END_GET
SET
                    lSuppress := Suppress;
                  
END_SET
END_PROPERTY

PROPERTY SuppressAfterCountDown : BOOL
GET
                    SuppressAfterCountDown := lSuppressAfterCountDown;
                  
END_GET
SET
                    lSuppressAfterCountDown := SuppressAfterCountDown;
                  
END_SET
END_PROPERTY

PROPERTY SupressCountDown : UINT
GET
                    SupressCountDown := lSupressCountDown;
                  
END_GET
SET
                    lSupressCountDown := SupressCountDown;
lResolvedSuppressAfterCountDown := FALSE;

IF (SupressCountDown>0) THEN
	lSuppressAfterCountDown := TRUE;
ELSE
	lSuppressAfterCountDown := FALSE;
END_IF

                  
END_SET
END_PROPERTY

PROPERTY TypeToken : t_medium_string
GET
                    TypeToken := 'Reportable';
                  
END_GET
END_PROPERTY
END_FUNCTION_BLOCK

FUNCTION_BLOCK ReportableSet
  VAR CONSTANT
    cReportableSetMax : USINT := 16;
  END_VAR
  VAR
    lMembers : t_reportable_array;
    lCount : USINT := 0;
    lDescribeFirstContextOnly : BOOL := FALSE;
  END_VAR

            
          

METHOD clear
                  lCount := 0;
                
END_METHOD

METHOD describe
  VAR_INPUT
    executeContext : POINTER TO ExecuteContext;
  END_VAR
  VAR
    i : USINT;
  END_VAR
                  IF (executeContext^.matchOption(cExecuteOptionSyntax)) THEN
	RETURN;
END_IF

IF (executeContext^.matchOption(cExecuteOptionParameter)) THEN	
	RETURN;
END_IF

executeContext^.append(', ');
executeContext^.WriteStream^.increaseIndent();
executeContext^.formatWithNewlineIndent();
executeContext^.append('"servers": [');
executeContext^.WriteStream^.increaseIndent();

FOR i:=1 TO Count DO	
	executeContext^.recordInitiatorWithNewlineIndent();
	lMembers[i]^.describe(executeContext);
	executeContext^.recordTerminator();

	IF (lDescribeFirstContextOnly) THEN
		EXIT;
	END_IF
	
	IF (i<Count) THEN
		executeContext^.append(', ');
	END_IF
END_FOR

executeContext^.WriteStream^.decreaseIndent();
executeContext^.append(']');
executeContext^.WriteStream^.decreaseIndent();

                
END_METHOD

METHOD equals
  VAR_INPUT
    source : POINTER TO ReportableSet;
  END_VAR
  VAR
    i : USINT;
  END_VAR
                  clear();

FOR i:=1 TO source^.Count DO
	lMembers[i] := source^.Members^[i];
END_FOR

lCount := source^.Count;

                
END_METHOD

METHOD initialize
                  lCount := 0;
                
END_METHOD

METHOD insert
  VAR_INPUT
    reportable : POINTER TO t_reportable;
  END_VAR
  VAR
    i : USINT;
    ptrA : POINTER TO POINTER TO t_reportable;
    ptrB : POINTER TO POINTER TO t_reportable;
  END_VAR
                  IF (reportable=0) THEN
	RETURN;
END_IF

IF (lCount>=cReportableSetMax) THEN
	RETURN;
END_IF

IF (lCount>0) THEN
	ptrA := ADR(lMembers[1]);
	ptrB := ADR(lMembers[2]);
	FOR i:=1 TO lCount DO
		ptrA^ := ptrB^;
		ptrA := ptrA + 1;
		ptrB := ptrB + 1;
	END_FOR
END_IF

lCount := lCount + 1;
lMembers[1] := reportable;

                
END_METHOD

METHOD list
  VAR_INPUT
    stream : POINTER TO t_stream;
  END_VAR
  VAR
    i : USINT;
  END_VAR
                  stream^.increaseIndent();

FOR i:=1 TO Count DO
	stream^.indent();
	stream^.append(lMembers[i]^.lIdentity);
	stream^.newline();
END_FOR

stream^.decreaseIndent();

                
END_METHOD

METHOD pop : POINTER TO t_reportable
                  IF (lCount=0) THEN
	pop := 0;
	RETURN;
END_IF

pop := lMembers[lCount];
lCount := lCount - 1;

                
END_METHOD

METHOD push
  VAR_INPUT
    reportable : POINTER TO t_reportable;
  END_VAR
                  IF (reportable=0) THEN
	RETURN;
END_IF

IF (lCount>=cReportableSetMax) THEN
	RETURN;
END_IF

lCount := lCount + 1;
lMembers[lCount] := reportable;
                
END_METHOD

METHOD replace
  VAR_INPUT
    reportable : POINTER TO t_reportable;
  END_VAR
                  clear();
push(reportable);
                
END_METHOD

PROPERTY Count : USINT
GET
                    Count := lCount;
                  
END_GET
END_PROPERTY

PROPERTY DescribeFirstContextOnly : BOOL
GET
                    DescribeFirstContextOnly := lDescribeFirstContextOnly;
                  
END_GET
SET
                    lDescribeFirstContextOnly := DescribeFirstContextOnly;
                  
END_SET
END_PROPERTY

PROPERTY Members : POINTER TO t_reportable_array
GET
                    Members := ADR(lMembers);
                  
END_GET
END_PROPERTY
END_FUNCTION_BLOCK

FUNCTION_BLOCK ReportableState EXTENDS Reportable
  VAR
    lVRLife : ValueReferenceUDINT;
    lLife : UDINT := 2;
    lCode : t_state_code;
    lExpiringChannelMask : UINT;
    lActive : BOOL := FALSE;
    lRegistered : BOOL := FALSE;
    lSuppressPrevious : BOOL := FALSE;
    lActiveRising : BOOL := FALSE;
    lUnsuppressRising : BOOL := FALSE;
    lUnsuppressFalling : BOOL := FALSE;
    lReportedInThisInstanceCount : UDINT := 0;
    lRaisedCount : UDINT := 0;  (* lUnsuppressedInThisInstanceCount: UDINT:= 0; *)
    lRaisedTimeStep : t_timestep := 0;
    lRaisedSystemTimeMicroseconds : ULINT := 0;
    lExpiresTimeStep : t_timestep;
    lSuppressUntilExpired : BOOL := FALSE;
    lSuppressAfterExpired : BOOL := FALSE;
    lContext : t_state_context := 0;
    lContextChanged : BOOL := FALSE;
  END_VAR

            
          

METHOD clear
                  Active := FALSE;
lContext := 0;

lExpiresTimeStep := gSystemServices.Cycle.TimeStep;

                
END_METHOD

METHOD describe
  VAR_INPUT
    executeContext : POINTER TO ExecuteContext;
  END_VAR
                  SUPER^.describe(executeContext);

IF (executeContext^.matchOption(cExecuteOptionSyntax)) THEN
	executeContext^.describeSyntaxExecutable(sCommandTrigger);
	RETURN;
END_IF

IF (executeContext^.matchOption(cExecuteOptionParameter)) THEN	
	RETURN;
END_IF

executeContext^.appendPair('style','state',TRUE,TRUE);

IF (lContext<>0) THEN
	executeContext^.appendPair('context',LWORD_TO_STRING(lContext),FALSE,TRUE);
END_IF

IF (executeContext^.matchOption(cExecuteOptionVerbose)) THEN	
	executeContext^.appendPair('raised',gTypeHandler.getTokenForUDINT(RaisedCount),FALSE,TRUE);
	executeContext^.appendPair('this_instance',gTypeHandler.getTokenForUDINT(ReportedInThisInstanceCount),FALSE,TRUE);
END_IF

                
END_METHOD

METHOD initialize
                  lVRLife.initializeValueReference(lLife,NopSelf,'Life','Duration of state once triggered','timestep',cValueStyleConfigurable);

SUPER^.initialize();

lActive := FALSE;
lRegistered := FALSE;
lRaisedCount := 0;
lRaisedTimeStep := 0;
lRaisedSystemTimeMicroseconds := 0;
lExpiresTimeStep := 0;

lChannelMask := gSystemServices.ReportableChannelManager.ChannelMaskDefaultState;


                
END_METHOD

METHOD initializeState
  VAR_INPUT
    p : POINTER TO t_particle_nop;
    nme : t_token_string;
    code : t_state_code;
  END_VAR
                  lCode := code;

IF (nme='') THEN
	Name := getStringForStateCode(Code);
ELSE
	Name := nme;
END_IF

IF (p=0) THEN
	gCodeErrorHandler(pMessage:='initializing reportable with null t_particle_nop');
	RETURN;
END_IF

p^.registerNonOperational(THIS);


                
END_METHOD

METHOD raise
                  lExpiresTimeStep := gSystemServices.Cycle.TimeStep + lLife;

lActiveRising := FALSE;
lUnsuppressRising := FALSE;
lUnsuppressFalling := FALSE;

// a := a+1;

IF (NOT(Active)) THEN
	Active := TRUE;
	lActiveRising := TRUE;
	
	lReportedInThisInstanceCount := 1;
	lRaisedCount := lRaisedCount + 1;
	lRaisedTimeStep := gSystemServices.Cycle.TimeStep;
	lRaisedSystemTimeMicroseconds := gSystemServices.Cycle.SystemTimeMicroseconds;

	IF (lSuppressUntilExpired) THEN
		SupressCountDown := 1; 	
	END_IF

	(*IF (Suppress) THEN
		lUnsuppressedInThisInstanceCount := 0;
	ELSE
		lUnsuppressedInThisInstanceCount := 1;	
	END_IF*)
	
	lSuppressPrevious := lSuppress;
	
	RETURN;
END_IF

lReportedInThisInstanceCount := lReportedInThisInstanceCount + 1;

IF ((NOT(lSuppressPrevious)) AND (lSuppress)) THEN
	lUnsuppressFalling := TRUE;
END_IF

IF ((NOT(lSuppress)) AND (lSuppressPrevious)) THEN
	lUnsuppressRising := TRUE;
END_IF

lSuppressPrevious := lSuppress;

(*IF (Suppress) THEN
	lUnsuppressedInThisInstanceCount := 0;
ELSE
	lUnsuppressedInThisInstanceCount := lUnsuppressedInThisInstanceCount + 1;	
END_IF*)

                
END_METHOD

METHOD report
  VAR_INPUT
    override : BOOL;
  END_VAR
                  IF ((override) OR 
	(Override)) THEN
	RETURN;
END_IF

SUPER^.report(override);

gSystemServices.ReportableChannelManager.reportState(THIS);
                
END_METHOD

METHOD trigger
  VAR_INPUT
    override : BOOL;
  END_VAR
                  IF (override) THEN
	RETURN;
END_IF 

report(FALSE);
propagate();

                
END_METHOD

METHOD triggerWithContext
  VAR_INPUT
    context : t_state_context;
  END_VAR
                  Context := context;
trigger(FALSE);

                
END_METHOD

METHOD execute
  VAR_INPUT
    executeContext : POINTER TO ExecuteContext;
  END_VAR
                  IF (executeContext^.matchCommand(sCommandTrigger)) THEN
	trigger(FALSE);
	RETURN;
END_IF

SUPER^.execute(executeContext);

                
END_METHOD

PROPERTY Active : BOOL
GET
                    Active := lActive;

                  
END_GET
SET
                    lActive := Active;
                  
END_SET
END_PROPERTY

PROPERTY ExpiringChannelMask : UINT
GET
                    ExpiringChannelMask := lExpiringChannelMask;
                  
END_GET
SET
                    lExpiringChannelMask := ExpiringChannelMask;
                  
END_SET
END_PROPERTY

PROPERTY Code : t_state_code
GET
                    Code := lCode;

                  
END_GET
SET
                    lCode:= Code;
                  
END_SET
END_PROPERTY

PROPERTY Context : t_state_context
GET
                    Context := lContext;
                  
END_GET
SET
                    IF (lContext=Context) THEN
	RETURN;
END_IF

lContext := Context;
lContextChanged := Active;

                  
END_SET
END_PROPERTY

PROPERTY ContextChanged : BOOL
GET
                    ContextChanged:= lContextChanged;
                  
END_GET
SET
                    lContextChanged := ContextChanged;
                  
END_SET
END_PROPERTY

PROPERTY ExpiresTimeStep : t_timestep
GET
                    ExpiresTimeStep := lExpiresTimeStep;
                  
END_GET
END_PROPERTY

PROPERTY Life : UDINT
GET
                    Life := lLife;

                  
END_GET
SET
                    lLife := MAX(Life,2);

                  
END_SET
END_PROPERTY

PROPERTY RaisedCount : UDINT
GET
                    RaisedCount := lRaisedCount;
                  
END_GET
END_PROPERTY

PROPERTY RaisedTimeStep : t_timestep
GET
                    RaisedTimeStep := lRaisedTimeStep;
                  
END_GET
END_PROPERTY

PROPERTY Registered : BOOL
GET
                    Registered := lRegistered;

                  
END_GET
SET
                    IF ((lRegistered) AND (NOT(Registered)) AND (SuppressAfterExpired)) THEN
	Suppress := TRUE;
END_IF

lRegistered := Registered;
                  
END_SET
END_PROPERTY

PROPERTY ReportedInThisInstanceCount : UDINT
GET
                    ReportedInThisInstanceCount := lReportedInThisInstanceCount;
                  
END_GET
END_PROPERTY

PROPERTY SuppressAfterExpired : BOOL
GET
                    SuppressAfterExpired := lSuppressAfterExpired;
                  
END_GET
SET
                    lSuppressAfterExpired := SuppressAfterExpired;
                  
END_SET
END_PROPERTY

PROPERTY SuppressUntilExpired : BOOL
GET
                    SuppressUntilExpired := lSuppressUntilExpired;
                  
END_GET
SET
                    IF ((lSuppressUntilExpired) AND (NOT(SuppressUntilExpired))) THEN
	SuppressAfterCountDown := FALSE;
END_IF

lSuppressUntilExpired := SuppressUntilExpired;

                  
END_SET
END_PROPERTY

PROPERTY TypeToken : t_medium_string
GET
                    TypeToken := 'State';
                  
END_GET
END_PROPERTY

PROPERTY ActiveRising : BOOL
GET
                    ActiveRising := lActiveRising;
                  
END_GET
END_PROPERTY

PROPERTY Suppress : BOOL
SET
                    lSuppress := Suppress;
                  
END_SET
END_PROPERTY

PROPERTY UnsuppressFalling : BOOL
GET
                    UnsuppressFalling := lUnsuppressFalling;

                  
END_GET
END_PROPERTY

PROPERTY UnsuppressRising : BOOL
GET
                    UnsuppressRising := lUnsuppressRising;
                  
END_GET
END_PROPERTY
END_FUNCTION_BLOCK

FUNCTION_BLOCK ReportableStateManager EXTENDS Particle
  VAR CONSTANT
    cCurrentMax : UINT := 255;
  END_VAR
  VAR
    lReportableChannelManager : POINTER TO ReportableChannelManager;
    lCurrent : ARRAY[1..cCurrentMax] OF POINTER TO t_reportablestate;
    lCurrentCount : UINT := 0;
    lOverflow : BOOL := FALSE;
    a : USINT := 0;
    b : USINT := 0;
  END_VAR

            
          

METHOD clear
  VAR_INPUT
    index : UINT;
  END_VAR
  VAR
    state : POINTER TO t_reportablestate;
    i : UINT;
  END_VAR
                  IF ((index=0) OR (index>lCurrentCount)) THEN
	RETURN;
END_IF

state := lCurrent[index];

lCurrentCount := lCurrentCount - 1;
FOR i:=index TO lCurrentCount DO
	lCurrent[i] := lCurrent[i+1];
END_FOR
lCurrent[lCurrentCount+1] := 0;

IF (state=0) THEN
	RETURN;
END_IF

state^.Registered := FALSE;
lReportableChannelManager^.reportStateExpired(state);
                
END_METHOD

METHOD cycle : POINTER TO t_reportableState
  VAR_INPUT
    mask : t_channel_mask;
    cycleIndex : POINTER TO UINT;
    loop : BOOL;
  END_VAR
  VAR
    count : UINT := 0;
    state : POINTER TO t_reportableState;
  END_VAR
                  IF ((lCurrentCount=0) OR 
	(cycleIndex=0)) THEN
	cycle := 0;
	RETURN;
END_IF

IF (cycleIndex^=0) THEN
	cycle := 0;
	RETURN;
END_IF

FOR count:=1 TO lCurrentCount DO
	IF (cycleIndex^>lCurrentCount) THEN
		IF (loop) THEN
			cycleIndex^ := 1;
		ELSE
			cycleIndex^ := 0;
			cycle := 0;
			RETURN;
		END_IF
	END_IF

	state := lCurrent[cycleIndex^]; // foobar assume state is non-null
	cycleIndex^ := cycleIndex^ + 1;
	
	IF ((NOT(state^.Suppress)) AND
		(NOT(state^.Override)) AND
		(fCheckChannelMask(state^.ChannelMask,mask))) THEN
		cycle := state;
		a := a+ 1;
		RETURN;
	END_IF
END_FOR

b := b+ 1;
cycleIndex^ := 0;
cycle := 0;
                
END_METHOD

METHOD describe
  VAR_INPUT
    executeContext : POINTER TO ExecuteContext;
  END_VAR
  VAR
    i : UINT;
    str : t_stream_string;
  END_VAR
                  SUPER^.describe(executeContext);

IF (executeContext^.matchOption(cExecuteOptionSyntax)) THEN
	RETURN;
END_IF

IF (executeContext^.matchOption(cExecuteOptionParameter)) THEN	
	RETURN;
END_IF

executeContext^.append(', ');
executeContext^.WriteStream^.increaseIndent();
executeContext^.formatWithNewlineIndent();
executeContext^.append('"states": [');
executeContext^.WriteStream^.increaseIndent();

FOR i:=1 TO lCurrentCount DO	
	executeContext^.recordInitiatorWithNewlineIndent();
	lCurrent[i]^.describe(executeContext);
	executeContext^.recordTerminator();
	
	IF (i<lCurrentCount) THEN
		executeContext^.append(', ');
	END_IF
END_FOR

executeContext^.WriteStream^.decreaseIndent();
executeContext^.append(']');
executeContext^.WriteStream^.decreaseIndent();

                
END_METHOD

METHOD initialize
  VAR
    i : UINT;
  END_VAR
                  IF (lReportableChannelManager=0) THEN
	gCodeErrorHandler(pMessage:=CONCAT('null pointer in ',lIdentity));
END_IF

SUPER^.initialize();

lCurrentCount := 0;
FOR i:=1 TO cCurrentMax DO
	lCurrent[i] := 0;
END_FOR

                
END_METHOD

METHOD initializeStateManager
  VAR_INPUT
    reportableChannelManager : POINTER TO ReportableChannelManager;
  END_VAR
                  lReportableChannelManager := reportableChannelManager;

                
END_METHOD

METHOD operator
  VAR
    i : UINT;
    state : POINTER TO t_reportablestate;
  END_VAR
                  FOR i:=1 TO lCurrentCount DO
	state := lCurrent[i];
	
	IF (state^.ContextChanged) THEN
		state^.ContextChanged := FALSE;
		lReportableChannelManager^.reportStateContextChanged(state);
	END_IF
	
	IF (state^.ExpiresTimeStep<=gSystemServices.Cycle.TimeStep) THEN
		clear(i);
	END_IF
END_FOR

                
END_METHOD

METHOD raise
  VAR_INPUT
    state : POINTER TO t_reportablestate;
  END_VAR
                  IF (state=0) THEN
	RETURN;
END_IF

IF (lCurrentCount>=cCurrentMax) THEN
	state^.Registered := FALSE;
	lOverflow := TRUE;
	RETURN;	
END_IF

IF (state^.Registered) THEN
	RETURN;
END_IF

lOverflow := FALSE;

lCurrentCount := lCurrentCount + 1;
lCurrent[lCurrentCount] := state;
state^.Registered := TRUE;

                
END_METHOD

PROPERTY Overflow : BOOL
GET
                    Overflow := lOverflow;
                  
END_GET
END_PROPERTY

PROPERTY TypeToken : t_medium_string
GET
                    TypeToken := 'RepStateManager';
                  
END_GET
END_PROPERTY
END_FUNCTION_BLOCK

FUNCTION fCheckUIRValidity : BOOL
  VAR_INPUT
    uir : REFERENCE TO t_ui_reportable;
  END_VAR

            IF (NOT(uir.valid)) THEN
	fCheckUIRValidity := FALSE;
	RETURN;
END_IF

IF ((uir.subsystem>cSubSystemMax) OR
	(uir.subsystem<0)) THEN
	fCheckUIRValidity := FALSE;
	RETURN;
END_IF

IF ((uir.event>cECMax) OR
	(uir.event<0)) THEN
	fCheckUIRValidity := FALSE;
	RETURN;
END_IF

IF ((uir.state>cSCMax) OR
	(uir.state<0)) THEN
	fCheckUIRValidity := FALSE;
	RETURN;
END_IF

fCheckUIRValidity := TRUE;

          
END_FUNCTION

FUNCTION getSeverityForStateCode : t_severity
  VAR_INPUT
    code : t_state_code;
  END_VAR

            getSeverityForStateCode := cSeverityNone; //foobar missing below

CASE code OF
	cSCNone:
		getSeverityForStateCode := cSeverityNone;

	cACSteerALargeSensorDelta:
		getSeverityForStateCode := cSeverityError;

	cACSecondaryNotRunning:
		getSeverityForStateCode := cSeverityError;

	cACSecondaryNotRunningModulation:
		getSeverityForStateCode := cSeverityError;

	cACSecondaryWaiting:
		getSeverityForStateCode := cSeverityWarning;

	cACSecondaryRunStateMismatch:
		getSeverityForStateCode := cSeverityWarning;

	cACSecondaryTemperature:
		getSeverityForStateCode := cSeverityWarning;
	
	cACChannelNotGood:
		getSeverityForStateCode := cSeverityError;

	cACChannelOperationalFail:
		getSeverityForStateCode := cSeverityError;

	cACChannelNotOperational:
		getSeverityForStateCode := cSeverityError;

	cACChannelOverflow:
		getSeverityForStateCode := cSeverityWarning;

	cACChannelSlaveFailed:
		getSeverityForStateCode := cSeverityError;

	cACCANOpenSlaveNotOperational:
		getSeverityForStateCode := cSeverityError;

	cACCANOpenSlaveModulation:
		getSeverityForStateCode := cSeverityError;

	cACCANOpenSlaveAllowableUp:
		getSeverityForStateCode := cSeverityError;

	cACCANOpenMasterNotOperational:
		getSeverityForStateCode := cSeverityError;

	cACCANOpenMasterModulation:
		getSeverityForStateCode := cSeverityError;

	cACCANOpenMasterAllowableUp:
		getSeverityForStateCode := cSeverityError;
	
	cACCANOpenSlaveNoValidTransmissions:
		getSeverityForStateCode := cSeverityWarning;

	cACCANOpenSlaveNotify:
		getSeverityForStateCode := cSeverityError;

	cACCANOpenSlaveBlock:
		getSeverityForStateCode := cSeverityError;

	cACCANOpenSlaveStop:
		getSeverityForStateCode := cSeverityCritical;
		
	cACUInterfaceEstop:
		getSeverityForStateCode := cSeverityCritical;

	cACUInterfaceStop:
		getSeverityForStateCode := cSeverityCritical;

	cACUInterfaceEmgy:
		getSeverityForStateCode := cSeverityWarning;

	cACUInterfaceNotReady:
		getSeverityForStateCode := cSeverityWarning;

	cACControllerTemperatureCutback:
		getSeverityForStateCode := cSeverityWarning;

	cACMotorTemperatureCutback:
		getSeverityForStateCode := cSeverityWarning;

	cACMotorTemperatureSensor:
		getSeverityForStateCode := cSeverityError;

	cACCoolantReservoir:
		getSeverityForStateCode := cSeverityWarning;

	cACCoolantTempHotCutback:
		getSeverityForStateCode := cSeverityWarning;

	cACCoolantTempColdCutback:
		getSeverityForStateCode := cSeverityWarning;

	cACCoolantHeating:
		getSeverityForStateCode := cSeverityError;

	cACCoolantChilling:
		getSeverityForStateCode := cSeverityError;

	cACCoolantSecondaryPowerFailHeatingCooling:
		getSeverityForStateCode := cSeverityError;

	cACCoolantSecondaryPowerFailPump:
		getSeverityForStateCode := cSeverityError;

	cACChargerOBCError:
		getSeverityForStateCode := cSeverityError;

	cACBMSAvailabilityInsufficient:
		getSeverityForStateCode := cSeverityError;

	cACBMSAvailabilityLimited:
		getSeverityForStateCode := cSeverityWarning;

	cBMSChargeAvailabilityLimited:
		getSeverityForStateCode := cSeverityWarning;

	cBMSChargeAvailabilityLimitedSevere:
		getSeverityForStateCode := cSeverityError;

	cBMSDischargeAvailabilityLimited:
		getSeverityForStateCode := cSeverityWarning;

	cBMSDischargeAvailabilityLimitedSevere:
		getSeverityForStateCode := cSeverityCritical;
		
	cACBMSRequestDisconnect:
		getSeverityForStateCode := cSeverityCritical;
	
	cACSOCBelowOperatingMinimum:
		getSeverityForStateCode := cSeverityError;

	cACSOCBelowStandbyMinimum:
		getSeverityForStateCode := cSeverityCritical;

	cACSOCWarningLow:
		getSeverityForStateCode := cSeverityWarning;
	
	cACBMSNotConnected:
		getSeverityForStateCode := cSeverityError;

	cACBMSChargeCutback:
		getSeverityForStateCode := cSeverityWarning;

	cACBMSDischargeCutback:
		getSeverityForStateCode := cSeverityWarning;

	cACBackupBatteryVoltageLow:
		getSeverityForStateCode := cSeverityError;

	cACBeaconsSecondaryPowerFail:
		getSeverityForStateCode := cSeverityError;

	cACSecondaryPowerFail:
		getSeverityForStateCode := cSeverityError;

	cACTMSStateMismatch:
		getSeverityForStateCode := cSeverityError;

	cACBMSChargeStateMismatch:
		getSeverityForStateCode := cSeverityError;

	cACBMSSOCMismatch:
		getSeverityForStateCode := cSeverityError;

	cACBMSVoltageMismatch:
		getSeverityForStateCode := cSeverityError;

	cACBMSCurrentMismatch:
		getSeverityForStateCode := cSeverityError;

	cACSensorRangeError:
		getSeverityForStateCode := cSeverityError;

	cACHydraulicFilter:
		getSeverityForStateCode := cSeverityError;

	cACHydraulicTemperature:
		getSeverityForStateCode := cSeverityWarning;
	
	cACBrakeLowHydraulicPressure:
		getSeverityForStateCode := cSeverityWarning;

	cACOutputFailure:
		getSeverityForStateCode := cSeverityError;
	
	cACDeviceTemperature:
		getSeverityForStateCode := cSeverityWarning;

	cACDeviceVoltage:
		getSeverityForStateCode := cSeverityWarning;

	cDCChargerStandby:
		getSeverityForStateCode := cSeverityNone;

	cDCChargerConnected:
		getSeverityForStateCode := cSeverityNone;

	cDCChargerDisconnected:
		getSeverityForStateCode := cSeverityNone;

	cDCTMSCooling:
		getSeverityForStateCode := cSeverityNone;

	cDCTMSHeating:
		getSeverityForStateCode := cSeverityNone;

	cDCBMSTMSCooling:
		getSeverityForStateCode := cSeverityNone;

	cDCBMSTMSHeating:
		getSeverityForStateCode := cSeverityNone;

	cDCBMSTMSNoCirculation:
		getSeverityForStateCode := cSeverityNone;

	cCCChargerStandby:
		getSeverityForStateCode := cSeverityNone;

	cCCChargerConnected:
		getSeverityForStateCode := cSeverityNone;

	cCCChargerDisconnected:
		getSeverityForStateCode := cSeverityNone;

	cCCWaitingForBrakeDisengaged:
		getSeverityForStateCode := cSeverityNone;

	cCCWaitingForParked:
		getSeverityForStateCode := cSeverityNone;

	cCCCommandStart:
		getSeverityForStateCode := cSeverityNone;

	cCCCommandStop:
		getSeverityForStateCode := cSeverityNone;

	cCCStopOnTimeout:
		getSeverityForStateCode := cSeverityNone;

	cCCLockoutInterlock:
		getSeverityForStateCode := cSeverityNone;

	cCCPosOnlyInterlock:
		getSeverityForStateCode := cSeverityNone;

	cCCScaledInterlock:
		getSeverityForStateCode := cSeverityNone;

	cCCThresholdInterlock:
		getSeverityForStateCode := cSeverityNone;

	cCCSynchronousInterlock:
		getSeverityForStateCode := cSeverityNone;

	cCCTwistlocksReadyInterlock:
		getSeverityForStateCode := cSeverityNone;
		
	cCCAutomaticStart:
		getSeverityForStateCode := cSeverityNone;
		
	cCCSyncState:
		getSeverityForStateCode := cSeverityNone;
		
	cCCCurrentUserNotEnabled:
		getSeverityForStateCode := cSeverityNone;
		
	cCCStandby:
		getSeverityForStateCode := cSeverityNone;
		
	cCCCycleOutput:
		getSeverityForStateCode := cSeverityNone;
END_CASE
          
END_FUNCTION

FUNCTION_BLOCK ReportableChannelUIRCache EXTENDS ReportableChannel
  VAR
    lUIRCacheManager : REFERENCE TO UIRCacheManager;
  END_VAR

            
          

METHOD _reportEvent
  VAR_INPUT
    event : POINTER TO t_reportableevent;
  END_VAR
  VAR
    uir : t_ui_reportable;
  END_VAR
                  uir.state := 0;
uir.event := event^.code;
uir.subsystem := event^.subsystem;
uir.active := TRUE;

lUIRCacheManager.reportUIR(uir);

                
END_METHOD

METHOD _reportStateExpired
  VAR_INPUT
    state : POINTER TO t_reportablestate;
  END_VAR
  VAR
    uir : t_ui_reportable;
  END_VAR
                  uir.state := state^.Code;
uir.event := 0;
uir.subsystem := state^.subsystem;
uir.active := FALSE;
	
lUIRCacheManager.reportUIR(uir);


                
END_METHOD

METHOD initialize
                  IF (NOT(__ISVALIDREF(lUIRCacheManager))) THEN
	gCodeErrorHandler(pMessage:=CONCAT('null reference in ',lIdentity));
END_IF

SUPER^.initialize();


                
END_METHOD

METHOD _reportState
  VAR_INPUT
    state : POINTER TO t_reportablestate;
    expired : BOOL;
  END_VAR
  VAR
    uir : t_ui_reportable;
  END_VAR
                  uir.state := state^.Code;
uir.event := 0;
uir.subsystem := state^.subsystem;
uir.active := NOT(expired);
	
lUIRCacheManager.reportUIR(uir);

                
END_METHOD

METHOD initializeUIRCache
  VAR_INPUT
    uIRCacheManager : REFERENCE TO UIRCacheManager;
  END_VAR
                  lUIRCacheManager REF= uIRCacheManager;

                
END_METHOD

METHOD _reportStateActiveRising
  VAR_INPUT
    state : POINTER TO t_reportablestate;
  END_VAR
                  _reportState(state);

                
END_METHOD

METHOD _reportStateUnsuppressFalling
  VAR_INPUT
    state : POINTER TO t_reportablestate;
  END_VAR
                  _reportStateExpired(state);

                
END_METHOD

METHOD _reportStateUnsuppressRising
  VAR_INPUT
    state : POINTER TO t_reportablestate;
  END_VAR
                  _reportState(state,FALSE);

                
END_METHOD

PROPERTY TypeToken : t_medium_string
GET
                    TypeToken := 'RepChanUIRCache';
                  
END_GET
END_PROPERTY
END_FUNCTION_BLOCK

FUNCTION_BLOCK UIRCacheManager EXTENDS OperationalParticleSet
  VAR
    lSubsystemCache : ARRAY[0..cSubsystemMax] OF UIRSubSystemCache;
    lReportedCount : UINT := 0;
  END_VAR

            
          

METHOD initialize
  VAR
    i : t_subsystem;
  END_VAR
                  FOR i:=0 TO cSubsystemMax DO
	lSubsystemCache[i].Name := gTypeHandler.getTokenForEnum(cEnumTypeSubsystem,i);
	registerOperational(ADR(lSubsystemCache[i]));	
END_FOR

SUPER^.initialize();

                
END_METHOD

METHOD reportUIR
  VAR_INPUT
    uir : t_ui_reportable;
  END_VAR
                  lSubsystemCache[uir.subsystem].reportUIR(uir);
lReportedCount := lReportedCount + 1;

                
END_METHOD

METHOD subsystemCache : REFERENCE TO UIRSubSystemCache
  VAR_INPUT
    i : t_subsystem;
  END_VAR
                  subsystemCache REF= lSubsystemCache[i];

                
END_METHOD

PROPERTY TypeToken : t_medium_string
GET
                    TypeToken := 'UIRCacheMgr';
                  
END_GET
END_PROPERTY
END_FUNCTION_BLOCK

FUNCTION_BLOCK UIREventCache EXTENDS Particle
  VAR
    lCache : ARRAY[1..cECMax] OF BOOL;
    lUpdated : BOOL := FALSE;
    lRefreshed : BOOL := FALSE;
    lSummaryStream : t_stream;
    lSummaryLines : t_summary_lines;
    lCount : USINT;
    lReportedCount : UINT := 0;
  END_VAR

            
          

METHOD reset
  VAR
    i : INT;
  END_VAR
                  FOR i:=1 TO cECMax DO
	lCache[i] := FALSE;
END_FOR

generateSummaryAndClear();

                
END_METHOD

METHOD initialize
                  SUPER^.initialize();

reset();

                
END_METHOD

METHOD generateSummaryAndClear
  VAR
    i : INT;
    count : USINT;
  END_VAR
                  lSummaryStream.clear();
lCount := 0;

FOR i:=1 TO cECMax DO
	IF (lCache[i]) THEN
		lSummaryStream.append(getStringForEventCode(i));
		lSummaryStream.newline();
		lCount := lCount + 1;

		IF (lCount<=cSummaryLines) THEN
			lSummaryLines[lCount] := getStringForEventCode(i);
		END_IF
		
		lCache[i] := FALSE;
	END_IF
END_FOR

IF (lCount>0) THEN
	lSummaryStream.append('total of <');
	lSummaryStream.append(USINT_TO_STRING(lCount));
	lSummaryStream.append('> events');
END_IF

FOR count:=lCount+1 TO cSummaryLines DO
	lSummaryLines[count] := '';
END_FOR

lRefreshed := TRUE;
                
END_METHOD

METHOD reportUIR
  VAR_INPUT
    uir : t_ui_reportable;
  END_VAR
                  lUpdated := ((lUpdated) OR (lCache[uir.event] <> uir.active));
lCache[uir.event] := uir.active;

lReportedCount := lReportedCount + 1;

                
END_METHOD

METHOD operator
                  SUPER^.operator();

lRefreshed := FALSE;

IF (lUpdated) THEN
	lUpdated := FALSE;
	
	generateSummaryAndClear();
END_IF


                
END_METHOD

PROPERTY SummaryStream : REFERENCE TO t_stream
SET
                    SummaryStream ref= lSummaryStream;

                  
END_SET
END_PROPERTY

PROPERTY Count : USINT
GET
                    Count:= lCount;
                  
END_GET
END_PROPERTY

PROPERTY Refreshed : BOOL
GET
                    Refreshed:= lRefreshed;
                  
END_GET
END_PROPERTY

PROPERTY SummaryLines : REFERENCE TO t_summary_lines
GET
                    SummaryLines ref= lSummaryLines;
                  
END_GET
END_PROPERTY

PROPERTY TypeToken : t_medium_string
GET
                    TypeToken := 'UIREventCache';
                  
END_GET
END_PROPERTY
END_FUNCTION_BLOCK

FUNCTION_BLOCK UIRRouter EXTENDS NonOperationalParticleSet
  VAR
    lReportableEvent : t_reportableevent;
    lReportableState : t_reportablestate;
  END_VAR

            
          

METHOD initialize
                  lReportableEvent.initializeEvent(NopSelf,'',cECNone);
lReportableState.initializeState(NopSelf,'',cSCNone);

SUPER^.initialize();

lReportableEvent.Suppress := FALSE;
lReportableEvent.ChannelMask := gSystemServices.ReportableChannelManager.ChannelMaskDefaultRoutedEvent;

lReportableState.Suppress := FALSE;
lReportableEvent.ChannelMask := gSystemServices.ReportableChannelManager.ChannelMaskDefaultRoutedState;

                
END_METHOD

METHOD reportUIR
  VAR_INPUT
    uir : t_ui_reportable;
  END_VAR
                  IF (uir.event>0) THEN
	lReportableEvent.Code := uir.event;
	lReportableEvent.ReportedTimeStep := gSystemServices.Cycle.TimeStep;

	IF (uir.active) THEN
		gSystemServices.ReportableChannelManager.routeEvent(ADR(lReportableEvent));
	END_IF
ELSIF (uir.state>0) THEN
	lReportableState.Code := uir.state;
	lReportableState.ReportedTimeStep := gSystemServices.Cycle.TimeStep;

	IF (uir.active) THEN
		gSystemServices.ReportableChannelManager.routeState(ADR(lReportableState));
	ELSE
		gSystemServices.ReportableChannelManager.routeStateExpired(ADR(lReportableState));
	END_IF
END_IF

                
END_METHOD

PROPERTY ReportableState : REFERENCE TO ReportableState
GET
                    ReportableState ref= lReportableState;
                  
END_GET
END_PROPERTY

PROPERTY ReportableEvent : REFERENCE TO ReportableEvent
GET
                    ReportableEvent ref= lReportableEvent;
                  
END_GET
END_PROPERTY

PROPERTY TypeToken : t_medium_string
GET
                    TypeToken := 'RepChanCache';
                  
END_GET
END_PROPERTY
END_FUNCTION_BLOCK

FUNCTION_BLOCK UIRStateCache EXTENDS Particle
  VAR
    lCache : ARRAY[1..cSCMax] OF BOOL;
    lUpdated : BOOL := FALSE;
    lRefreshed : BOOL := FALSE;
    lSummaryStream : t_stream;
    lSummaryLines : t_summary_lines;
    lCount : USINT;
    lSeverity : t_severity;
    lReportedCount : UINT := 0;
  END_VAR

            
          

METHOD reset
  VAR
    i : t_state_code;
  END_VAR
                  FOR i:=1 TO cSCMax DO
	lCache[i] := FALSE;
END_FOR

generateSummary();

                
END_METHOD

METHOD reportUIR
  VAR_INPUT
    uir : t_ui_reportable;
  END_VAR
                  lUpdated := ((lUpdated) OR (lCache[uir.state] <> uir.active));
lCache[uir.state] := uir.active;

lReportedCount := lReportedCount + 1;

                
END_METHOD

METHOD initialize
                  SUPER^.initialize();

reset();

                
END_METHOD

METHOD operator
                  SUPER^.operator();

lRefreshed := FALSE;

IF (lUpdated) THEN
	lUpdated := FALSE;
	
	generateSummary();
END_IF
                
END_METHOD

METHOD generateSummary
  VAR
    i : t_state_code;
    count : USINT;
  END_VAR
                  lSummaryStream.clear();
lCount := 0;
lSeverity := cSeverityNone;

FOR i:=1 TO cSCMax DO
	IF (lCache[i]) THEN
		lSummaryStream.append(getStringForStateCode(i));
		lSummaryStream.newline();
		
		lCount := lCount + 1;

		IF (lCount<=cSummaryLines) THEN
			lSummaryLines[lCount] := getStringForStateCode(i);
		END_IF
	
		lSeverity := MAX(lSeverity,getSeverityForStateCode(i));
	END_IF
END_FOR

IF (lCount>0) THEN
	lSummaryStream.append('total of <');
	lSummaryStream.append(USINT_TO_STRING(lCount));
	lSummaryStream.append('> alarms with highest severity <');
	lSummaryStream.append(gTypeHandler.getTokenForEnum(cEnumTypeSeverity,lSeverity));
	lSummaryStream.append('>');
END_IF

FOR count:=lCount+1 TO cSummaryLines DO
	lSummaryLines[count] := '';
END_FOR

lRefreshed := TRUE;
                
END_METHOD

PROPERTY SummaryStream : REFERENCE TO t_stream
GET
                    SummaryStream ref= lSummaryStream;
                  
END_GET
END_PROPERTY

PROPERTY Count : USINT
GET
                    Count:= lCount;
                  
END_GET
END_PROPERTY

PROPERTY Refreshed : BOOL
GET
                    Refreshed:= lRefreshed;
                  
END_GET
END_PROPERTY

PROPERTY TypeToken : t_medium_string
GET
                    TypeToken := 'UIRStateCache';
                  
END_GET
END_PROPERTY

PROPERTY Severity : t_severity
GET
                    Severity := lSeverity;
                  
END_GET
END_PROPERTY

PROPERTY SummaryLines : REFERENCE TO t_summary_lines
GET
                    SummaryLines ref= lSummaryLines;
                  
END_GET
END_PROPERTY
END_FUNCTION_BLOCK

FUNCTION_BLOCK UIRSubSystemCache EXTENDS OperationalParticleSet
  VAR
    lEventCache : UIREventCache;
    lStateCache : UIRStateCache;
    lReportedCount : UINT := 0;
  END_VAR

            
          

METHOD reset
                  lEventCache.reset();
lStateCache.reset();

                
END_METHOD

METHOD reportUIR
  VAR_INPUT
    uir : t_ui_reportable;
  END_VAR
                  IF (uir.event>0) THEN
	lEventCache.reportUIR(uir);
ELSE
	lStateCache.reportUIR(uir);
END_IF

lReportedCount := lReportedCount + 1;


                
END_METHOD

METHOD initialize
                  registerOperational(ADR(lEventCache));
registerOperational(ADR(lStateCache));

SUPER^.initialize();



                
END_METHOD

PROPERTY EventCache : REFERENCE TO UIREventCache
GET
                    EventCache ref= lEventCache;
                  
END_GET
END_PROPERTY

PROPERTY StateCache : REFERENCE TO UIRStateCache
GET
                    StateCache ref= lStateCache;
                  
END_GET
END_PROPERTY

PROPERTY TypeToken : t_medium_string
GET
                    TypeToken := 'UIRSubSysCache';
                  
END_GET
END_PROPERTY
END_FUNCTION_BLOCK

FUNCTION_BLOCK ReportableChargeModulation EXTENDS ReportableState
  VAR
    lQualifier : t_charge_qualifier;
    lScalingCharge : t_percentage;
    lScalingDischarge : t_percentage;
    lThresholdCharge : t_percentage;
    lThresholdDischarge : t_percentage;
    lServers : ARRAY[1..16] OF POINTER TO ReportableContextChargeModulation;
    lServerCount : USINT := 0;
  END_VAR

            
          

METHOD clear
                  lQualifier := cChargeQualifierNone;
lScalingCharge := 1.0;
lScalingDischarge := 1.0;
lThresholdCharge := 1.0;
lThresholdDischarge := 1.0;

SUPER^.clear();
                
END_METHOD

METHOD describe
  VAR_INPUT
    executeContext : POINTER TO ExecuteContext;
  END_VAR
  VAR
    i : USINT;
  END_VAR
                  SUPER^.describe(executeContext);

IF (executeContext^.matchOption(cExecuteOptionSyntax)) THEN
	RETURN;
END_IF

IF (executeContext^.matchOption(cExecuteOptionParameter)) THEN	
	RETURN;
END_IF

IF (executeContext^.matchOption(cExecuteOptionVerbose)) THEN	
	executeContext^.appendPair('qualifier',gTypeHandler.getTokenForEnum(cEnumTypeChargeQualifier,Qualifier),TRUE,TRUE);
	executeContext^.appendPair('scaling_charge',gTypeHandler.getTokenForPercentage(ScalingCharge),TRUE,TRUE);
	executeContext^.appendPair('scaling_discharge',gTypeHandler.getTokenForPercentage(ScalingDischarge),TRUE,TRUE);
	executeContext^.appendPair('threshold_charge',gTypeHandler.getTokenForPercentage(ThresholdCharge),TRUE,TRUE);
	executeContext^.appendPair('threshold_discharge',gTypeHandler.getTokenForPercentage(ThresholdDischarge),TRUE,TRUE);
END_IF

executeContext^.append(', "servers": [');

FOR i:=1 TO lServerCount DO	
	executeContext^.appendIdentity(lServers[i]);
	
	IF (i<>lServerCount) THEN
		executeContext^.append(', ');
	END_IF
END_FOR

executeContext^.append(']');


                
END_METHOD

METHOD pause
                  lQualifier := cChargeQualifierBoth;
lScalingCharge :=0.0;
lScalingDischarge :=0.0;
lThresholdCharge :=0.0;
lThresholdDischarge :=0.0;

                
END_METHOD

METHOD propagate
  VAR
    i : USINT;
  END_VAR
                  lPropagateCount := lPropagateCount + 1;

FOR i:=1 TO lServerCount DO
	lServers[i]^.processReportableChargeModulation(THIS,FALSE);
END_FOR
                
END_METHOD

METHOD registerServer
  VAR_INPUT
    server : POINTER TO ReportableContextChargeModulation;
  END_VAR
  VAR
    i : USINT;
  END_VAR
                  IF (server=0) THEN
	RETURN;
END_IF

IF (lServerCount>=16) THEN
	gCodeErrorHandler(pMessage:='Reportable register overflow');
	RETURN;
END_IF

FOR i:=1 TO lServerCount DO
	IF (lServers[i]=server) THEN
		RETURN;
	END_IF
END_FOR

lServerCount := lServerCount + 1;
lServers[lServerCount] := server;

                
END_METHOD

PROPERTY Qualifier : t_charge_qualifier
GET
                    Qualifier := lQualifier;
                  
END_GET
SET
                    lQualifier := Qualifier;

                  
END_SET
END_PROPERTY

PROPERTY ScalingCharge : t_percentage
GET
                    ScalingCharge := lScalingCharge;
                  
END_GET
SET
                    lScalingCharge := abs(ScalingCharge);
                  
END_SET
END_PROPERTY

PROPERTY ScalingDischarge : t_percentage
GET
                    ScalingDischarge := lScalingDischarge;
                  
END_GET
SET
                    lScalingDischarge := abs(ScalingDischarge);
                  
END_SET
END_PROPERTY

PROPERTY ThresholdCharge : t_percentage
GET
                    ThresholdCharge := lThresholdCharge;
                  
END_GET
SET
                    lThresholdCharge := abs(ThresholdCharge);
                  
END_SET
END_PROPERTY

PROPERTY ThresholdDischarge : t_percentage
GET
                    ThresholdDischarge := lThresholdDischarge;
                  
END_GET
SET
                    lThresholdDischarge := abs(ThresholdDischarge);
                  
END_SET
END_PROPERTY

PROPERTY TypeToken : t_medium_string
GET
                    TypeToken := 'ChargeMod';
                  
END_GET
END_PROPERTY
END_FUNCTION_BLOCK

FUNCTION_BLOCK ReportableContextChargeModulation EXTENDS ReportableContextEvent
  VAR
    lQualifier : PendingChargeQualifier;
    lScalingCharge : PendingPercentage;
    lScalingDischarge : PendingPercentage;
    lThresholdCharge : PendingPercentage;
    lThresholdDischarge : PendingPercentage;
  END_VAR

            
          

METHOD describe
  VAR_INPUT
    executeContext : POINTER TO ExecuteContext;
  END_VAR
                  SUPER^.describe(executeContext);

IF (executeContext^.matchOption(cExecuteOptionSyntax)) THEN
	RETURN;
END_IF

IF (executeContext^.matchOption(cExecuteOptionParameter)) THEN	
	RETURN;
END_IF

IF (executeContext^.matchOption(cExecuteOptionVerbose)) THEN	
	executeContext^.appendPair('qualifier',gTypeHandler.getTokenForEnum(cEnumTypeChargeQualifier,Qualifier),TRUE,TRUE);
	executeContext^.appendPair('scaling_charge',gTypeHandler.getTokenForPercentage(ScalingCharge),TRUE,TRUE);
	executeContext^.appendPair('scaling_discharge',gTypeHandler.getTokenForPercentage(ScalingDischarge),TRUE,TRUE);
	executeContext^.appendPair('threshold_charge',gTypeHandler.getTokenForPercentage(ThresholdCharge),TRUE,TRUE);
	executeContext^.appendPair('threshold_discharge',gTypeHandler.getTokenForPercentage(ThresholdDischarge),TRUE,TRUE);
END_IF

                
END_METHOD

METHOD operator
                  lQualifier.operator(Override);
lScalingCharge.operator(Override);
lScalingDischarge.operator(Override);
lThresholdCharge.operator(Override);
lThresholdDischarge.operator(Override);

SUPER^.operator();

                
END_METHOD

METHOD processReportableChargeModulation
  VAR_INPUT
    reportable : POINTER TO ReportableChargeModulation;
    override : BOOL;
  END_VAR
                  IF (reportable=0) THEN
	RETURN;
END_IF

IF (reportable^.Qualifier=cChargeQualifierNone) THEN
	RETURN;
END_IF

lPendingContext.push(reportable);

IF ((override) OR
	(reportable^.Override)) THEN
	IncludesOverrides := true;
	RETURN;
END_IF

Qualifier := reportable^.Qualifier;
	
CASE reportable^.Qualifier OF
	cChargeQualifierBoth:
		ScalingCharge := reportable^.ScalingCharge;
		ScalingDischarge := reportable^.ScalingDischarge;
		ThresholdCharge := reportable^.ThresholdCharge;
		ThresholdDischarge := reportable^.ThresholdDischarge;
						
	cChargeQualifierCharge:
		ScalingCharge := reportable^.ScalingCharge;
		ThresholdCharge := reportable^.ThresholdCharge;

	cChargeQualifierDischarge:
		ScalingDischarge := reportable^.ScalingDischarge;
		ThresholdDischarge := reportable^.ThresholdDischarge;
END_CASE

                
END_METHOD

PROPERTY Qualifier : t_charge_qualifier
GET
                    Qualifier := lQualifier.Value;
                  
END_GET
SET
                    lQualifier.Pending := Qualifier;

                  
END_SET
END_PROPERTY

PROPERTY ScalingCharge : t_percentage
GET
                    ScalingCharge := lScalingCharge.Value;
                  
END_GET
SET
                    lScalingCharge.Pending := ScalingCharge;
                  
END_SET
END_PROPERTY

PROPERTY ScalingDischarge : t_percentage
GET
                    ScalingDischarge := lScalingDischarge.Value;
                  
END_GET
SET
                    lScalingDischarge.Pending := ScalingDischarge;
                  
END_SET
END_PROPERTY

PROPERTY ThresholdCharge : t_percentage
GET
                    ThresholdCharge := lThresholdCharge.Value;
                  
END_GET
SET
                    lThresholdCharge.Pending := ThresholdCharge;
                  
END_SET
END_PROPERTY

PROPERTY ThresholdDischarge : t_percentage
GET
                    ThresholdDischarge := lThresholdDischarge.Value;
                  
END_GET
SET
                    lThresholdDischarge.Pending := ThresholdDischarge;
                  
END_SET
END_PROPERTY

PROPERTY TypeToken : t_medium_string
GET
                    TypeToken := 'CntxtQualMod';
                  
END_GET
END_PROPERTY
END_FUNCTION_BLOCK

FUNCTION_BLOCK ReportableContextChargeModulationRCSM EXTENDS ReportableContextChargeModulation
  VAR
    lPositiveIsCharge : BOOL := FALSE;
    lNegativeIsCharge : BOOL := FALSE;
    lServers : ARRAY[1..16] OF POINTER TO ReportableContextSignedModulation;
    lServerCount : USINT := 0;
  END_VAR

            
          

METHOD describe
  VAR_INPUT
    executeContext : POINTER TO ExecuteContext;
  END_VAR
  VAR
    i : USINT;
  END_VAR
                  SUPER^.describe(executeContext);

IF (executeContext^.matchOption(cExecuteOptionSyntax)) THEN
	RETURN;
END_IF

IF (executeContext^.matchOption(cExecuteOptionParameter)) THEN
	RETURN;
END_IF

executeContext^.append(', "servers": [');

FOR i:=1 TO lServerCount DO
	executeContext^.appendIdentity(lServers[i]);
	
	IF (i<>lServerCount) THEN
		executeContext^.append(', ');
	END_IF
END_FOR

executeContext^.append(']');

                
END_METHOD

METHOD initializeEvent
  VAR_INPUT
    p : POINTER TO t_particle_nop;
    name : t_token_string;
    code : t_event_code;
  END_VAR
                  SUPER^.initializeEvent(p,name,code);

lContext.initialize();
lPendingContext.initialize();

lIncludesOverrides.Default := FALSE;

                
END_METHOD

METHOD propagate
  VAR
    i : USINT;
    interlockSt : t_interlock_state := cInterlockStateWarning;  (* assume that the is some modulation so at least a warning *)
    scalingPos : t_percentage := 1.0;
    scalingNeg : t_percentage := 1.0;
    thresholdPos : t_percentage := 1.0;
    thresholdNeg : t_percentage := 1.0;
  END_VAR
                  lPropagateCount := lPropagateCount + 1;

IF (lPositiveIsCharge) THEN
	scalingPos := ScalingCharge;
	thresholdPos := ThresholdCharge;	
ELSE
	scalingPos := ScalingDischarge;
	thresholdPos := ThresholdDischarge;		
END_IF

IF (lNegativeIsCharge) THEN
	scalingNeg := ScalingCharge;
	thresholdNeg:=ThresholdCharge;
ELSE
	scalingNeg := ScalingDischarge;
	thresholdNeg := ThresholdDischarge;	
END_IF

IF ((scalingPos=0.0) OR (thresholdPos=0.0)) THEN
	interlockSt := cInterlockStateErrorPositive;
END_IF
IF ((scalingNeg=0.0) OR (thresholdNeg=0.0)) THEN
	IF (interlockSt=cInterlockStateErrorPositive) THEN
		interlockSt := cInterlockStateError;
	ELSE
		interlockSt := cInterlockStateErrorNegative;		
	END_IF
END_IF

FOR i:=1 TO lServerCount DO
	lServers[i]^.processReportable(THIS,FALSE,
		interlockSt,
		scalingPos,
		scalingNeg,
		thresholdPos,
		thresholdNeg);
END_FOR

                
END_METHOD

METHOD registerServer
  VAR_INPUT
    server : POINTER TO ReportableContextSignedModulation;
  END_VAR
  VAR
    i : USINT;
  END_VAR
                  IF (server=0) THEN
	RETURN;
END_IF

IF (lServerCount>=16) THEN
	gCodeErrorHandler(pMessage:='Reportable register overflow');
	RETURN;
END_IF

FOR i:=1 TO lServerCount DO
	IF (lServers[i]=server) THEN
		RETURN;
	END_IF
END_FOR

lServerCount := lServerCount + 1;
lServers[lServerCount] := server;

                
END_METHOD

PROPERTY NegativeIsCharge : BOOL
GET
                    NegativeIsCharge := lNegativeIsCharge;
                  
END_GET
SET
                    lNegativeIsCharge := NegativeIsCharge;
                  
END_SET
END_PROPERTY

PROPERTY PositiveIsCharge : BOOL
GET
                    PositiveIsCharge := lPositiveIsCharge;
                  
END_GET
SET
                    lPositiveIsCharge := PositiveIsCharge;
                  
END_SET
END_PROPERTY

PROPERTY TypeToken : t_medium_string
GET
                    TypeToken := 'CntxtQualModEx';
                  
END_GET
END_PROPERTY
END_FUNCTION_BLOCK

FUNCTION_BLOCK ReportableContextEvent EXTENDS ReportableEvent
  VAR
    lContext : t_reportable_set;
    lPendingContext : t_reportable_set;
    lIncludesOverrides : PendingBool;
  END_VAR

            
          

METHOD describe
  VAR_INPUT
    executeContext : POINTER TO ExecuteContext;
  END_VAR
                  SUPER^.describe(executeContext);

IF (executeContext^.matchOption(cExecuteOptionSyntax)) THEN
	RETURN;
END_IF

IF (executeContext^.matchOption(cExecuteOptionParameter)) THEN	
	RETURN;
END_IF

IF (executeContext^.matchOption(cExecuteOptionVerbose)) THEN	
	executeContext^.appendPair('includes_overrides',gTypeHandler.getTokenForBool(IncludesOverrides),FALSE,TRUE);
END_IF

executeContext^.append(', "context": ');	
lContext.describe(executeContext);

                
END_METHOD

METHOD initializeEvent
  VAR_INPUT
    p : POINTER TO t_particle_nop;
    name : t_token_string;
    code : t_event_code;
  END_VAR
                  SUPER^.initializeEvent(p,name,code);

lContext.initialize();
lPendingContext.initialize();

lIncludesOverrides.Default := FALSE;

                
END_METHOD

METHOD operator
                  lContext.equals(ADR(lPendingContext));
lPendingContext.clear();

lIncludesOverrides.operator(FALSE);

IF (lContext.Count<>0) THEN
	report(FALSE);
	propagate();
END_IF


                
END_METHOD

METHOD reportIfContext
  VAR_INPUT
    override : BOOL;
  END_VAR
                  IF (lContext.Count=0) THEN
	RETURN;
END_IF

report(override);
                
END_METHOD

PROPERTY Context : POINTER TO t_reportable_set
GET
                    Context := ADR(lContext);
                  
END_GET
END_PROPERTY

PROPERTY IncludesOverrides : BOOL
GET
                    IncludesOverrides := lIncludesOverrides.Value;
                  
END_GET
SET
                    lIncludesOverrides.Pending := IncludesOverrides;
                  
END_SET
END_PROPERTY

PROPERTY PendingContext : POINTER TO t_reportable_set
GET
                    PendingContext := ADR(lPendingContext);
                  
END_GET
END_PROPERTY

PROPERTY TypeToken : t_medium_string
GET
                    TypeToken := 'ContextEvent';
                  
END_GET
END_PROPERTY
END_FUNCTION_BLOCK

FUNCTION_BLOCK ReportableContextSignedModulation EXTENDS ReportableContextEvent
  VAR
    lInterlockState : PendingInterlockState;
    lScalingPositive : PendingPercentage;
    lScalingNegative : PendingPercentage;
    lThresholdPositive : PendingPercentage;
    lThresholdNegative : PendingPercentage;
    lProcessCount : USINT;
    lProcessSignedModulationCount : USINT;
  END_VAR

            
          

METHOD describe
  VAR_INPUT
    executeContext : POINTER TO ExecuteContext;
  END_VAR
                  SUPER^.describe(executeContext);

IF (executeContext^.matchOption(cExecuteOptionSyntax)) THEN
	RETURN;
END_IF

IF (executeContext^.matchOption(cExecuteOptionParameter)) THEN	
	RETURN;
END_IF

IF (executeContext^.matchOption(cExecuteOptionVerbose)) THEN	
	executeContext^.appendPair('interlock_state',gTypeHandler.getTokenForEnum(cEnumTypeInterlockState,InterlockState),TRUE,TRUE);
	executeContext^.appendPair('scaling_positive',gTypeHandler.getTokenForPercentage(ScalingPositive),TRUE,TRUE);
	executeContext^.appendPair('scaling_negative',gTypeHandler.getTokenForPercentage(ScalingNegative),TRUE,TRUE);
	executeContext^.appendPair('threshold_positive',gTypeHandler.getTokenForPercentage(ThresholdPositive),TRUE,TRUE);
	executeContext^.appendPair('threshold_negative',gTypeHandler.getTokenForPercentage(ThresholdNegative),TRUE,TRUE);
END_IF

                
END_METHOD

METHOD operator
                  lInterlockState.operator(Override);
lScalingPositive.operator(Override);
lScalingNegative.operator(Override);
lThresholdPositive.operator(Override);
lThresholdNegative.operator(Override);

SUPER^.operator();

                
END_METHOD

METHOD processReportable
  VAR_INPUT
    reportable : POINTER TO t_reportable;
    override : BOOL;
    interlockSt : t_interlock_state;
    scalingPos : t_percentage;
    scalingNeg : t_percentage;
    thresholdPos : t_percentage;
    thresholdNeg : t_percentage;
  END_VAR
                  IF (reportable=0) THEN
	RETURN;
END_IF

IF (interlockSt=cInterlockStateNone) THEN
	RETURN;
END_IF

lPendingContext.push(reportable);

IF ((override) OR
	(reportable^.Override)) THEN
	IncludesOverrides := true;
	RETURN;
END_IF

lProcessCount := lProcessCount + 1;

InterlockState := interlockSt;
ScalingPositive := scalingPos;
ScalingNegative := scalingNeg;
ThresholdPositive := thresholdPos;
ThresholdNegative := thresholdNeg;

                
END_METHOD

METHOD processReportableSignedModulation
  VAR_INPUT
    reportable : POINTER TO ReportableSignedModulation;
    override : BOOL;
  END_VAR
                  IF (reportable=0) THEN
	RETURN;
END_IF

IF (reportable^.InterlockState=cInterlockStateNone) THEN
	RETURN;
END_IF

lPendingContext.push(reportable);

IF ((override) OR
	(reportable^.Override)) THEN
	IncludesOverrides := true;
	RETURN;
END_IF

lProcessSignedModulationCount := lProcessSignedModulationCount + 1;

InterlockState := reportable^.InterlockState;
ScalingPositive := reportable^.ScalingPositive;
ScalingNegative := reportable^.ScalingNegative;
ThresholdPositive := reportable^.ThresholdPositive;
ThresholdNegative := reportable^.ThresholdNegative;

                
END_METHOD

METHOD stop : t_percentage
  VAR_INPUT
    value : t_percentage;
  END_VAR
                  stop := 0.0;

                
END_METHOD

METHOD update : t_percentage
  VAR_INPUT
    value : t_percentage;
  END_VAR
                  IF (Override) THEN
	update := value;
	RETURN;
END_IF

IF (lContext.Count=0) THEN
	update := value;
	RETURN;	
END_IF

IF ((InterlockState>=cInterlockStateOveride) OR
	(InterlockState=cInterlockStateNone) OR
	(InterlockState=cInterlockStateGood)) THEN
	update := value;
	RETURN;
END_IF

IF (InterlockState<=cInterlockStateError) THEN
	update := stop(value);
	RETURN;
END_IF

IF (value<0) THEN
	update := MAX(value*ScalingNegative,-1.0*ABS(ThresholdNegative));
ELSIF (value>0) THEN
	update := MIN(value*ScalingPositive,ABS(ThresholdPositive));
ELSE
	update := value;
END_IF

                
END_METHOD

PROPERTY InterlockState : t_interlock_state
GET
                    InterlockState := lInterlockState.Value;
                  
END_GET
SET
                    lInterlockState.Pending := InterlockState;
                  
END_SET
END_PROPERTY

PROPERTY ScalingNegative : t_percentage
GET
                    ScalingNegative := lScalingNegative.Value;
                  
END_GET
SET
                    lScalingNegative.Pending := ScalingNegative;
                  
END_SET
END_PROPERTY

PROPERTY ScalingPositive : t_percentage
GET
                    ScalingPositive := lScalingPositive.Value;
                  
END_GET
SET
                    lScalingPositive.Pending := ScalingPositive;
                  
END_SET
END_PROPERTY

PROPERTY ThresholdNegative : t_percentage
GET
                    ThresholdNegative := lThresholdNegative.Value;
                  
END_GET
SET
                    lThresholdNegative.Pending := ThresholdNegative;

                  
END_SET
END_PROPERTY

PROPERTY ThresholdPositive : t_percentage
GET
                    ThresholdPositive := lThresholdPositive.Value;
                  
END_GET
SET
                    lThresholdPositive.Pending := ThresholdPositive;

                  
END_SET
END_PROPERTY

PROPERTY TypeToken : t_medium_string
GET
                    TypeToken := 'CntxtSgnMod';
                  
END_GET
END_PROPERTY
END_FUNCTION_BLOCK

FUNCTION_BLOCK ReportableSignedModulation EXTENDS ReportableState
  VAR
    lInterlockState : t_interlock_state := cInterlockStateGood;
    lScalingPositive : t_percentage;
    lScalingNegative : t_percentage;
    lThresholdPositive : t_percentage;
    lThresholdNegative : t_percentage;
    lServers : ARRAY[1..16] OF POINTER TO ReportableContextSignedModulation;
    lServerCount : USINT := 0;
  END_VAR

            
          

METHOD clear
                  lInterlockState := cInterlockStateGood;
lScalingPositive := 1.0;
lScalingNegative := 1.0;
lThresholdPositive := 1.0;
lThresholdNegative := 1.0;

SUPER^.clear();
                
END_METHOD

METHOD describe
  VAR_INPUT
    executeContext : POINTER TO ExecuteContext;
  END_VAR
  VAR
    i : USINT;
  END_VAR
                  SUPER^.describe(executeContext);

IF (executeContext^.matchOption(cExecuteOptionSyntax)) THEN
	RETURN;
END_IF

IF (executeContext^.matchOption(cExecuteOptionParameter)) THEN
	RETURN;
END_IF

IF (executeContext^.matchOption(cExecuteOptionVerbose)) THEN	
	executeContext^.appendPair('interlock_state',gTypeHandler.getTokenForEnum(cEnumTypeInterlockState,InterlockState),TRUE,TRUE);
	executeContext^.appendPair('scaling_positive',gTypeHandler.getTokenForPercentage(ScalingPositive),TRUE,TRUE);
	executeContext^.appendPair('scaling_negative',gTypeHandler.getTokenForPercentage(ScalingNegative),TRUE,TRUE);
	executeContext^.appendPair('threshold_positive',gTypeHandler.getTokenForPercentage(ThresholdPositive),TRUE,TRUE);
	executeContext^.appendPair('threshold_negative',gTypeHandler.getTokenForPercentage(ThresholdNegative),TRUE,TRUE);
END_IF

executeContext^.append(', "servers": [');

FOR i:=1 TO lServerCount DO
	executeContext^.appendIdentity(lServers[i]);

	IF (i<>lServerCount) THEN
		executeContext^.append(', ');
	END_IF
END_FOR

executeContext^.append(']');

                
END_METHOD

METHOD pause
                  lInterlockState := cInterlockStateError;
lScalingPositive :=0.0;
lScalingNegative :=0.0;
lThresholdPositive :=0.0;
lThresholdNegative :=0.0;
                
END_METHOD

METHOD propagate
  VAR
    i : USINT;
  END_VAR
                  lPropagateCount := lPropagateCount + 1;

FOR i:=1 TO lServerCount DO
	lServers[i]^.processReportableSignedModulation(THIS,FALSE);
END_FOR
                
END_METHOD

METHOD registerServer
  VAR_INPUT
    server : POINTER TO ReportableContextSignedModulation;
  END_VAR
  VAR
    i : USINT;
  END_VAR
                  IF (server=0) THEN
	RETURN;
END_IF

IF (lServerCount>=16) THEN
	gCodeErrorHandler(pMessage:='Reportable register overflow');
	RETURN;
END_IF

FOR i:=1 TO lServerCount DO
	IF (lServers[i]=server) THEN
		RETURN;
	END_IF
END_FOR

lServerCount := lServerCount + 1;
lServers[lServerCount] := server;

                
END_METHOD

PROPERTY InterlockState : t_interlock_state
GET
                    InterlockState := lInterlockState;
                  
END_GET
SET
                    lInterlockState := InterlockState;
                  
END_SET
END_PROPERTY

PROPERTY ScalingNegative : t_percentage
GET
                    ScalingNegative := lScalingNegative;
                  
END_GET
SET
                    lScalingNegative := ScalingNegative;
                  
END_SET
END_PROPERTY

PROPERTY ScalingPositive : t_percentage
GET
                    ScalingPositive := lScalingPositive;
                  
END_GET
SET
                    lScalingPositive := ScalingPositive;
                  
END_SET
END_PROPERTY

PROPERTY ThresholdNegative : t_percentage
GET
                    ThresholdNegative := lThresholdNegative;
                  
END_GET
SET
                    lThresholdNegative := ThresholdNegative;
                  
END_SET
END_PROPERTY

PROPERTY ThresholdPositive : t_percentage
GET
                    ThresholdPositive := lThresholdPositive;
                  
END_GET
SET
                    lThresholdPositive := ThresholdPositive;
                  
END_SET
END_PROPERTY

PROPERTY TypeToken : t_medium_string
GET
                    TypeToken := 'SgnMod';
                  
END_GET
END_PROPERTY
END_FUNCTION_BLOCK

FUNCTION_BLOCK ReportableContextSystemControl EXTENDS ReportableContextEvent
  VAR
    lControl : PendingSystemControl;
    lAllowableSystemState : PendingSystemStateUp;
  END_VAR

            
          

METHOD describe
  VAR_INPUT
    executeContext : POINTER TO ExecuteContext;
  END_VAR
                  SUPER^.describe(executeContext);

IF (executeContext^.matchOption(cExecuteOptionSyntax)) THEN
	RETURN;
END_IF

IF (executeContext^.matchOption(cExecuteOptionParameter)) THEN	
	RETURN;
END_IF

executeContext^.appendPair('control',gTypeHandler.getTokenForEnum(cEnumTypeSystemControl,Control),TRUE,TRUE);

IF (executeContext^.matchOption(cExecuteOptionVerbose)) THEN	
	executeContext^.appendPair('allowable_system_state',gTypeHandler.getTokenForEnum(cEnumTypeSystemState,AllowableSystemState),TRUE,TRUE);
END_IF

                
END_METHOD

METHOD apply
                  IF (Control=cSystemControlReset) THEN
	IF (gSystemServices.SystemState.State>cSystemStatePreOperational) THEN
		gSystemServices.SystemState.transitionStop(cSystemStatePreOperational,THIS,Override);
	ELSE
		gSystemServices.SystemState.transitionInitialized(AllowableSystemState,THIS,Override);		
	END_IF
	
	RETURN;
END_IF

IF (Control=cSystemControlEstop) THEN
	gSystemServices.SystemState.transitionEstop(AllowableSystemState,THIS,Override);
	RETURN;
END_IF

IF (Control=cSystemControlStop) THEN
	gSystemServices.SystemState.transitionStop(AllowableSystemState,THIS,Override);
	RETURN;
END_IF

IF (Control=cSystemControlStart) THEN
	gSystemServices.SystemState.transitionStart(AllowableSystemState,THIS,Override);
	RETURN;
END_IF

                
END_METHOD

METHOD operator
                  lControl.operator(Override);
lAllowableSystemState.operator(Override);

SUPER^.operator();

                
END_METHOD

METHOD processReportableSystemControl
  VAR_INPUT
    reportable : POINTER TO ReportableSystemControl;
    override : BOOL;
  END_VAR
                  IF (reportable=0) THEN
	RETURN;
END_IF

IF (reportable^.Control=cSystemControlNone) THEN
	RETURN;
END_IF

IF ((override) OR
	(reportable^.Override)) THEN
	IncludesOverrides := TRUE;
	lPendingContext.push(reportable);	
	RETURN;
END_IF

IF (reportable^.Control<lControl.Pending) THEN
	lPendingContext.insert(reportable);
ELSE
	lPendingContext.push(reportable);	
END_IF

Control := reportable^.Control;
AllowableSystemState := reportable^.AllowableSystemState;

                
END_METHOD

PROPERTY AllowableSystemState : t_system_state
GET
                    AllowableSystemState := lAllowableSystemState.Value;
                  
END_GET
SET
                    lAllowableSystemState.Pending := AllowableSystemState;
                  
END_SET
END_PROPERTY

PROPERTY Control : t_system_control
GET
                    Control := lControl.Value;
                  
END_GET
SET
                    lControl.Pending := Control;
                  
END_SET
END_PROPERTY

PROPERTY TypeToken : t_medium_string
GET
                    TypeToken := 'CntxtSysCntrl';
                  
END_GET
END_PROPERTY
END_FUNCTION_BLOCK

FUNCTION_BLOCK ReportableSystemControl EXTENDS ReportableState
  VAR
    lControl : t_system_control;
    lAllowableSystemState : t_system_state;
  END_VAR

            
          

METHOD describe
  VAR_INPUT
    executeContext : POINTER TO ExecuteContext;
  END_VAR
                  SUPER^.describe(executeContext);

IF (executeContext^.matchOption(cExecuteOptionSyntax)) THEN
	RETURN;
END_IF

IF (executeContext^.matchOption(cExecuteOptionParameter)) THEN	
	RETURN;
END_IF

executeContext^.appendPair('control',gTypeHandler.getTokenForEnum(cEnumTypeSystemControl,Control),TRUE,TRUE);
executeContext^.appendPair('allowable_system_state',gTypeHandler.getTokenForEnum(cEnumTypeSystemState,AllowableSystemState),TRUE,TRUE);


                
END_METHOD

METHOD propagate
                  lPropagateCount := lPropagateCount + 1;

gSystemServices.SystemState.SystemControl.processReportableSystemControl(THIS,FALSE);

                
END_METHOD

METHOD initialize
                  SUPER^.initialize();

lSuppress := FALSE;

                
END_METHOD

PROPERTY AllowableSystemState : t_system_state
GET
                    AllowableSystemState := lAllowableSystemState;
                  
END_GET
SET
                    lAllowableSystemState := AllowableSystemState;
                  
END_SET
END_PROPERTY

PROPERTY Control : t_system_control
GET
                    Control := lControl;
                  
END_GET
SET
                    lControl := Control;
                  
END_SET
END_PROPERTY

PROPERTY TypeToken : t_medium_string
GET
                    TypeToken := 'SysCntrl';
                  
END_GET
END_PROPERTY
END_FUNCTION_BLOCK

FUNCTION_BLOCK ReportableContextSystemState EXTENDS ReportableContextEvent
  VAR
    lUpdateState : ValueObjectEnumType;
  END_VAR

            
          

METHOD describe
  VAR_INPUT
    executeContext : POINTER TO ExecuteContext;
  END_VAR
                  SUPER^.describe(executeContext);

IF (executeContext^.matchOption(cExecuteOptionSyntax)) THEN
	RETURN;
END_IF

IF (executeContext^.matchOption(cExecuteOptionParameter)) THEN	
	RETURN;
END_IF

executeContext^.appendPair('state',gTypeHandler.getTokenForEnum(cEnumTypeSystemState,State),TRUE,TRUE);

                
END_METHOD

METHOD check : t_system_state
  VAR_INPUT
    stte : t_system_state;
  END_VAR
                  IF (lPendingContext.Count=0) THEN
	check := stte;
	RETURN;
END_IF

check := Pending;

                
END_METHOD

METHOD initialize
                  lUpdateState.EnumType := cEnumTypeSystemState;
lUpdateState.initializeValueObject(NopSelf,'UpdateState','Updated state','',cValueStyleConfigurable);

SUPER^.initialize();

                
END_METHOD

METHOD process
  VAR_INPUT
    stte : t_system_state;
    reportable : POINTER TO t_reportable;
    override : BOOL;
  END_VAR
                  IF (reportable=0) THEN
	RETURN;
END_IF

lPendingContext.push(reportable);

IF ((override) OR
	(reportable^.Override)) THEN
	IncludesOverrides := true;
	RETURN;
END_IF

State := stte;

                
END_METHOD

METHOD updatex : t_system_state
  VAR_INPUT
    stte : t_system_state;
  END_VAR
                  IF (OverrideUpdate) THEN
	update := lOverrideUpdateState;
	RETURN;
END_IF

IF ((lContext.Count=0) OR
	(Override)) THEN
	update := stte;
	RETURN;
END_IF

update := State;

                
END_METHOD

METHOD update : t_system_state
  VAR_INPUT
    stte : t_system_state;
  END_VAR
                  IF ((lContext.Count=0) OR
	(Override)) THEN
	lUpdateState.Value := stte;
ELSE
	lUpdateState.Value := State;
END_IF

lUpdateState.operator();
update := lUpdateState.Value;

                
END_METHOD

PROPERTY Pending : t_system_state
GET
                    Pending := cSystemStateNone;
                  
END_GET
END_PROPERTY

PROPERTY State : t_system_state
GET
                    State := cSystemStateNone;

                  
END_GET
SET
                    ;

                  
END_SET
END_PROPERTY

PROPERTY TypeToken : t_medium_string
GET
                    TypeToken := 'CntxtSysState';
                  
END_GET
END_PROPERTY
END_FUNCTION_BLOCK

FUNCTION_BLOCK ReportableContextSystemStateDown EXTENDS ReportableContextSystemState
  VAR
    lState : PendingSystemStateDown;
  END_VAR

            
          

METHOD operator
                  lState.operator(Override);

SUPER^.operator();

                
END_METHOD

PROPERTY Pending : t_system_state
GET
                    Pending := lState.Pending;
                  
END_GET
END_PROPERTY

PROPERTY State : t_system_state
GET
                    State := lState.Value;

                  
END_GET
SET
                    lState.Pending := State;

                  
END_SET
END_PROPERTY

PROPERTY TypeToken : t_medium_string
GET
                    TypeToken := 'CntxtSysStateDn';
                  
END_GET
END_PROPERTY
END_FUNCTION_BLOCK

FUNCTION_BLOCK ReportableContextSystemStateUp EXTENDS ReportableContextSystemState
  VAR
    lState : PendingSystemStateUp;
  END_VAR

            
          

METHOD operator
                  lState.operator(Override);

SUPER^.operator();

                
END_METHOD

PROPERTY Pending : t_system_state
GET
                    Pending := lState.Pending;
                  
END_GET
END_PROPERTY

PROPERTY State : t_system_state
GET
                    State := lState.Value;

                  
END_GET
SET
                    lState.Pending := State;

                  
END_SET
END_PROPERTY

PROPERTY TypeToken : t_medium_string
GET
                    TypeToken := 'CntxtSysStateUp';
                  
END_GET
END_PROPERTY
END_FUNCTION_BLOCK

FUNCTION_BLOCK ReportableSystemStateTransition EXTENDS ReportableContextEvent
  VAR
    lCurrentState : t_system_state;
    lNextState : t_system_state;
  END_VAR

            
          

METHOD describe
  VAR_INPUT
    executeContext : POINTER TO ExecuteContext;
  END_VAR
                  SUPER^.describe(executeContext);

IF (executeContext^.matchOption(cExecuteOptionSyntax)) THEN
	RETURN;
END_IF

IF (executeContext^.matchOption(cExecuteOptionParameter)) THEN	
	RETURN;
END_IF

executeContext^.appendPair('state',gTypeHandler.getTokenForEnum(cEnumTypeSystemState,NextState),TRUE,TRUE);


                
END_METHOD

METHOD initialize
                  SUPER^.initialize();

lSuppress := FALSE;

                
END_METHOD

PROPERTY NextState : t_system_state
GET
                    NextState := lNextState;

                  
END_GET
SET
                    lNextState := NextState;

                  
END_SET
END_PROPERTY

PROPERTY TypeToken : t_medium_string
GET
                    TypeToken := 'CntxtSysStTrans';
                  
END_GET
END_PROPERTY
END_FUNCTION_BLOCK

FUNCTION_BLOCK ReportableContextModulation EXTENDS ReportableContextEvent
  VAR
    lScaling : PendingPercentage;
    lThreshold : PendingPercentage;
  END_VAR

            
          

METHOD describe
  VAR_INPUT
    executeContext : POINTER TO ExecuteContext;
  END_VAR
                  SUPER^.describe(executeContext);

IF (executeContext^.matchOption(cExecuteOptionSyntax)) THEN
	RETURN;
END_IF

IF (executeContext^.matchOption(cExecuteOptionParameter)) THEN	
	RETURN;
END_IF

IF (executeContext^.matchOption(cExecuteOptionVerbose)) THEN	
	executeContext^.appendPair('scaling',gTypeHandler.getTokenForPercentage(Scaling),TRUE,TRUE);
	executeContext^.appendPair('threshold',gTypeHandler.getTokenForPercentage(Threshold),TRUE,TRUE);
END_IF


                
END_METHOD

METHOD operator
                  lScaling.operator(Override);
lThreshold.operator(Override);

SUPER^.operator();

                
END_METHOD

METHOD processReportableModulation
  VAR_INPUT
    reportable : POINTER TO ReportableModulation;
    override : BOOL;
  END_VAR
                  IF (reportable=0) THEN
	RETURN;
END_IF

lPendingContext.push(reportable);

IF ((override) OR
	(reportable^.Override)) THEN
	IncludesOverrides := true;
	RETURN;
END_IF

Scaling := reportable^.Scaling;
Threshold := reportable^.Threshold;

                
END_METHOD

PROPERTY Scaling : t_percentage
GET
                    Scaling := lScaling.Value;
                  
END_GET
SET
                    lScaling.Pending := Scaling;

                  
END_SET
END_PROPERTY

PROPERTY Threshold : t_percentage
GET
                    Threshold := lThreshold.Value;

                  
END_GET
SET
                    lThreshold.Pending := Threshold;
                  
END_SET
END_PROPERTY

PROPERTY TypeToken : t_medium_string
GET
                    TypeToken := 'CntxtMod';
                  
END_GET
END_PROPERTY
END_FUNCTION_BLOCK

FUNCTION_BLOCK ReportableModulation EXTENDS ReportableState
  VAR
    lScaling : t_percentage;
    lThreshold : t_percentage;
  END_VAR

            
          

METHOD describe
  VAR_INPUT
    executeContext : POINTER TO ExecuteContext;
  END_VAR
                  SUPER^.describe(executeContext);

IF (executeContext^.matchOption(cExecuteOptionSyntax)) THEN
	RETURN;
END_IF

IF (executeContext^.matchOption(cExecuteOptionParameter)) THEN	
	RETURN;
END_IF

IF (executeContext^.matchOption(cExecuteOptionVerbose)) THEN	
	executeContext^.appendPair('scaling',gTypeHandler.getTokenForPercentage(Scaling),TRUE,TRUE);
	executeContext^.appendPair('threshold',gTypeHandler.getTokenForPercentage(Threshold),TRUE,TRUE);
END_IF


                
END_METHOD

METHOD pause
                  lScaling :=0.0;
lThreshold :=0.0;


                
END_METHOD

PROPERTY Scaling : t_percentage
GET
                    Scaling := lScaling;
                  
END_GET
SET
                    lScaling := abs(Scaling);
                  
END_SET
END_PROPERTY

PROPERTY Threshold : t_percentage
GET
                    Threshold := lThreshold;
                  
END_GET
SET
                    lThreshold := abs(Threshold);
                  
END_SET
END_PROPERTY

PROPERTY TypeToken : t_medium_string
GET
                    TypeToken := 'Mod';
                  
END_GET
END_PROPERTY
END_FUNCTION_BLOCK

FUNCTION_BLOCK ParticleReporterEvent EXTENDS ReportableEvent
  VAR CONSTANT
    cReportableParticleSetMax : USINT := 64;
  END_VAR
  VAR
    lTimer : t_timer;
    lReportableParticleCount : USINT := 0;
    lReportableParticleSet : ARRAY[1..64] OF t_particle_ptr;
  END_VAR

            
          

METHOD initialize
                  SUPER^.initialize();

lTimer.initialize();
lTimer.Enable := TRUE;
lTimer.Period := T#1M;

lSuppress := FALSE;

lChannelMask := gSystemServices.ReportableChannelManager.ChannelMaskDefaultParticleReporterEvent;


                
END_METHOD

METHOD execute
  VAR_INPUT
    executeContext : POINTER TO ExecuteContext;
  END_VAR
  VAR
    token : t_token_string;
    particle : t_particle_ptr;
    index : UINT;
    i : UINT;
    id : UINT;
  END_VAR
                  IF (executeContext^.matchCommand(sCommandRegister)) THEN
	IF (NOT(executeContext^.configureUINT(cTokenObject,id,TRUE,THIS))) THEN
		RETURN;
	END_IF

	particle := gSystemServices.getParticle(token,id);
	IF (particle=0) THEN
		executeContextFail(executeContext,cExecuteReturnUnknownArgumentValue,TRUE);
		RETURN;		
	END_IF

	IF (findParticle(particle)>0) THEN
		RETURN;
	END_IF
	
	IF (lReportableParticleCount>=cReportableParticleSetMax) THEN
		executeContextFail(executeContext,cExecuteReturnSetOverflow,TRUE);
		RETURN;
	END_IF

	lReportableParticleCount := lReportableParticleCount + 1;
	lReportableParticleSet[lReportableParticleCount] := particle;

	RETURN;
END_IF

IF (executeContext^.matchCommand(sCommandClear)) THEN
	
	FOR i:=1 TO lReportableParticleCount DO
		lReportableParticleSet[i] := 0;
	END_FOR
	lReportableParticleCount := 0;

	RETURN;
END_IF

IF (executeContext^.matchCommand(sCommandDeregister)) THEN
	IF (NOT(executeContext^.configureUINT(cTokenObject,id,TRUE,THIS))) THEN
		RETURN;
	END_IF
	
	particle := gSystemServices.getParticle(token,id);
	IF (particle=0) THEN
		executeContextFail(executeContext,cExecuteReturnUnknownArgumentValue,TRUE);
		RETURN;		
	END_IF

	index := findParticle(particle);
	IF (index=0) THEN
		RETURN;
	END_IF

	lReportableParticleCount := lReportableParticleCount - 1;	
	FOR i:=index TO lReportableParticleCount DO
		lReportableParticleSet[i] := lReportableParticleSet[i+1];
	END_FOR
	lReportableParticleSet[lReportableParticleCount+1] := 0;

	RETURN;
END_IF

SUPER^.execute(executeContext);

                
END_METHOD

METHOD operator
                  lTimer.operator();
IF (lTimer.Expired) THEN
	lTimer.reset();
	
	IF (lReportableParticleCount>0) THEN
		trigger(FALSE);
	END_IF
END_IF

SUPER^.operator();
                
END_METHOD

METHOD findParticle : USINT
  VAR_INPUT
    particle : t_particle_ptr;
  END_VAR
  VAR
    i : USINT;
  END_VAR
                  FOR i:=1 TO lReportableParticleCount DO
	IF (lReportableParticleSet[i]=particle) THEN
		findParticle := i;
		RETURN;
	END_IF
END_FOR

findParticle := 0;

                
END_METHOD

METHOD describe
  VAR_INPUT
    executeContext : POINTER TO ExecuteContext;
  END_VAR
  VAR
    i : USINT;
  END_VAR
                  SUPER^.describe(executeContext);

IF (executeContext^.matchOption(cExecuteOptionSyntax)) THEN
	executeContext^.describeSyntaxExecutable(sCommandRegister);
	executeContext^.describeSyntaxExecutable(sCommandClear);
	executeContext^.describeSyntaxExecutable(sCommandDeregister);

	RETURN;
END_IF

IF (executeContext^.matchOption(cExecuteOptionParameter)) THEN
	RETURN;
END_IF

executeContext^.append(', ');
executeContext^.WriteStream^.increaseIndent();
executeContext^.formatWithNewlineIndent();
executeContext^.append('"members": [');
executeContext^.WriteStream^.increaseIndent();

FOR i:=1 TO lReportableParticleCount DO	
	executeContext^.recordInitiatorWithNewlineIndent();
	lReportableParticleSet[i]^.describe(executeContext);
	executeContext^.recordTerminator();
	
	IF (i<lReportableParticleCount) THEN
		executeContext^.append(', ');
	END_IF
END_FOR

executeContext^.WriteStream^.decreaseIndent();
executeContext^.append(']');
executeContext^.WriteStream^.decreaseIndent();

                
END_METHOD

PROPERTY TypeToken : t_medium_string
GET
                    TypeToken := 'ParticleRepEvent';
                  
END_GET
END_PROPERTY

PROPERTY Period : t_time
GET
                    Period := lTimer.Period;
                  
END_GET
SET
                    lTimer.Period := Period;
                  
END_SET
END_PROPERTY
END_FUNCTION_BLOCK

FUNCTION_BLOCK ReportableAlarm EXTENDS ReportableState
  VAR
    lSeverity : t_severity := cSeverityWarning;
    lState : BOOL := FALSE;
    lInputReference : REFERENCE TO UINT;
    lMask : WORD;
    lTriggerInput : WORD;
  END_VAR

            
          

METHOD describe
  VAR_INPUT
    executeContext : POINTER TO ExecuteContext;
  END_VAR
                  SUPER^.describe(executeContext);

IF (executeContext^.matchOption(cExecuteOptionSyntax)) THEN
	RETURN;
END_IF

IF (executeContext^.matchOption(cExecuteOptionParameter)) THEN	
	RETURN;
END_IF

executeContext^.appendPair('alarm_state',gTypeHandler.getTokenForUSINT(BOOL_TO_USINT(lActive)),FALSE,TRUE);
executeContext^.appendPair('severity',gTypeHandler.getTokenForEnum(cEnumTypeSeverity,Severity),TRUE,TRUE);

IF (executeContext^.matchOption(cExecuteOptionVerbose)) THEN	
	executeContext^.appendPair('input',gTypeHandler.getTokenForUINT(lInputReference),FALSE,TRUE);
	executeContext^.appendPair('mask',WORD_TO_STRING(Mask),FALSE,TRUE);
	executeContext^.appendPair('state',gTypeHandler.getTokenForBool(State),FALSE,TRUE);
END_IF

                
END_METHOD

METHOD initializeStateOp
  VAR_INPUT
    p : POINTER TO t_particle_op;
    name : t_token_string;
    code : t_state_code;
  END_VAR
                  lCode := code;

IF (name='') THEN
	Name := getStringForStateCode(Code);
ELSE
	Name := name;
END_IF

IF (p=0) THEN
	gCodeErrorHandler(pMessage:='initializing reportable with null t_particle_op');
	RETURN;
END_IF

p^.registerOperational(THIS);


                
END_METHOD

METHOD operator
                  IF (NOT(__ISVALIDREF(lInputReference))) THEN
	RETURN;
END_IF

lState := WORD_TO_BOOL(lMask AND UINT_TO_WORD(lInputReference));

SUPER^.operator();

IF (lState) THEN
	lTriggerInput := UINT_TO_WORD(lInputReference);
	trigger(FALSE);
END_IF

                
END_METHOD

METHOD initialize
                  SUPER^.initialize();

lSuppress := FALSE;

                
END_METHOD

PROPERTY InputReference : REFERENCE TO UINT
SET
                    lInputReference REF= InputReference;


                  
END_SET
END_PROPERTY

PROPERTY Mask : WORD
GET
                    Mask := lMask;
                  
END_GET
SET
                    lMask := Mask;
                  
END_SET
END_PROPERTY

PROPERTY Severity : t_severity
GET
                    Severity := lSeverity;
                  
END_GET
SET
                    lSeverity := Severity;
                  
END_SET
END_PROPERTY

PROPERTY State : BOOL
GET
                    State := lState;
                  
END_GET
END_PROPERTY

PROPERTY TypeToken : t_medium_string
GET
                    TypeToken := 'Alarm';
                  
END_GET
END_PROPERTY
END_FUNCTION_BLOCK

FUNCTION_BLOCK ReportableAlarmAllowableUp EXTENDS ReportableAlarmEscalating
  VAR
    lAllowableSystemState : t_system_state := cSystemStateGoOperational;
    lUpperSystemStateScope : t_system_state := cSystemStateGoOperational;
    lLowerSystemStateScope : t_system_state := cSystemStateGoOperational;
    lForceTrigger : BOOL := FALSE;
  END_VAR

            
          

METHOD describe
  VAR_INPUT
    executeContext : POINTER TO ExecuteContext;
  END_VAR
                  SUPER^.describe(executeContext);

IF (executeContext^.matchOption(cExecuteOptionSyntax)) THEN
	RETURN;
END_IF

IF (executeContext^.matchOption(cExecuteOptionParameter)) THEN	
	RETURN;
END_IF

IF (executeContext^.matchOption(cExecuteOptionVerbose)) THEN	
	executeContext^.appendPair('allowable',gTypeHandler.getTokenForEnum(cEnumTypeSystemState,AllowableSystemState),TRUE,TRUE);
END_IF


                
END_METHOD

METHOD test
  VAR_INPUT
    override : BOOL;
  END_VAR
                  IF (override) THEN
	RETURN;
END_IF

IF ((gSystemServices.SystemState.State>lUpperSystemStateScope) OR
	(gSystemServices.SystemState.State<lLowerSystemStateScope)) THEN
	IF ((lForceTrigger) AND
		(Severity>cSeverityNone)) THEN
		trigger(FALSE);
	END_IF

	RETURN;	
END_IF

trigger(FALSE);

gSystemServices.SystemState.transitionAllowUp(lAllowableSystemState,THIS,Override);

                
END_METHOD

PROPERTY AllowableSystemState : t_system_state
GET
                    AllowableSystemState := lAllowableSystemState;
                  
END_GET
SET
                    lAllowableSystemState := AllowableSystemState;
                  
END_SET
END_PROPERTY

PROPERTY ForceTrigger : BOOL
GET
                    ForceTrigger := lForceTrigger;
                  
END_GET
SET
                    lForceTrigger := ForceTrigger;
                  
END_SET
END_PROPERTY

PROPERTY LowerSystemStateScope : t_system_state
GET
                    LowerSystemStateScope := lLowerSystemStateScope;
                  
END_GET
SET
                    lLowerSystemStateScope := LowerSystemStateScope;
                  
END_SET
END_PROPERTY

PROPERTY TypeToken : t_medium_string
GET
                    TypeToken := 'AlarmAllowUp';
                  
END_GET
END_PROPERTY

PROPERTY UpperSystemStateScope : t_system_state
GET
                    UpperSystemStateScope := lUpperSystemStateScope;
                  
END_GET
SET
                    lUpperSystemStateScope := UpperSystemStateScope;
                  
END_SET
END_PROPERTY
END_FUNCTION_BLOCK

FUNCTION_BLOCK ReportableAlarmEscalating EXTENDS ReportableAlarm
  VAR CONSTANT
    cSeverityWarningThreshold : ULINT := 500000;
    cSeverityErrorThreshold : ULINT := 2000000;
    cSeverityCriticalThreshold : ULINT := 8000000;
    cSeverityWarningTimeout : t_time := TIME#500ms;
    cSeverityErrorTimeout : t_time := TIME#2s0ms;
    cSeverityCriticalTimeout : t_time := TIME#8s0ms;
  END_VAR
  VAR
    lInitialSeverity : t_severity := cSeverityNone;
    lSeverityWarningThreshold : ULINT := cSeverityWarningThreshold;
    lSeverityErrorThreshold : ULINT := cSeverityErrorThreshold;
    lSeverityCriticalThreshold : ULINT := cSeverityCriticalThreshold;
    lSeverityWarningTimeout : t_time := cSeverityWarningTimeout;
    lSeverityErrorTimeout : t_time := cSeverityErrorTimeout;
    lSeverityCriticalTimeout : t_time := cSeverityCriticalTimeout;
  END_VAR

            
          

METHOD calibrate
  VAR
    averageCycleTime : ULINT := 32000;
  END_VAR
                  lSeverityErrorTimeout := MAX(lSeverityWarningTimeout,lSeverityErrorTimeout);
lSeverityCriticalTimeout := MAX(lSeverityErrorTimeout,lSeverityCriticalTimeout);

lSeverityWarningThreshold := TIME_TO_ULINT(lSeverityWarningTimeout);
lSeverityErrorThreshold := TIME_TO_ULINT(lSeverityErrorTimeout);
lSeverityCriticalThreshold := TIME_TO_ULINT(lSeverityCriticalTimeout);

                
END_METHOD

METHOD initializeState
  VAR_INPUT
    p : POINTER TO t_particle_nop;
    nme : t_token_string;
    code : t_state_code;
  END_VAR
                  SUPER^.initializeState(p,nme,code);

calibrate();

                
END_METHOD

METHOD report
  VAR_INPUT
    override : BOOL;
  END_VAR
  VAR
    systemTimeMicroseconds : ULINT;
    duration : ULINT;
  END_VAR
                  IF ((override) OR 
	(Override)) THEN
	Severity := InitialSeverity;
	RETURN;
END_IF

IF (NOT(Active)) THEN
	Severity := InitialSeverity;	
END_IF

SUPER^.report(override);

systemTimeMicroseconds := gSystemServices.Cycle.SystemTimeMicroseconds;
IF (systemTimeMicroseconds>lRaisedSystemTimeMicroseconds) THEN
	duration := systemTimeMicroseconds - lRaisedSystemTimeMicroseconds;
ELSE
	duration := 0;
END_IF

CASE Severity OF
	cSeverityNone:
		IF (duration>lSeverityWarningThreshold) THEN
			Severity := cSeverityWarning;
		END_IF
		
	cSeverityWarning:
		IF (duration>lSeverityErrorThreshold) THEN
			Severity := cSeverityError;
		END_IF
	
	cSeverityError:
		IF (duration>lSeverityCriticalThreshold) THEN
			Severity := cSeverityCritical;
		END_IF
END_CASE

                
END_METHOD

PROPERTY InitialSeverity : t_severity
GET
                    InitialSeverity := lInitialSeverity;
                  
END_GET
SET
                    lInitialSeverity := InitialSeverity;
                  
END_SET
END_PROPERTY

PROPERTY SeverityCriticalTimeout : t_time
GET
                    SeverityCriticalTimeout := lSeverityCriticalTimeout;
                  
END_GET
SET
                    lSeverityCriticalTimeout := SeverityCriticalTimeout;

calibrate();
                  
END_SET
END_PROPERTY

PROPERTY SeverityErrorTimeout : t_time
GET
                    SeverityErrorTimeout := lSeverityErrorTimeout;
                  
END_GET
SET
                    lSeverityErrorTimeout := SeverityErrorTimeout;

calibrate();
                  
END_SET
END_PROPERTY

PROPERTY SeverityWarningTimeout : t_time
GET
                    SeverityWarningTimeout := lSeverityWarningTimeout;
                  
END_GET
SET
                    lSeverityWarningTimeout := SeverityWarningTimeout;

calibrate();
                  
END_SET
END_PROPERTY

PROPERTY TypeToken : t_medium_string
GET
                    TypeToken := 'EscAlarm';
                  
END_GET
END_PROPERTY
END_FUNCTION_BLOCK

FUNCTION_BLOCK ReportableAlarmMaskReferenceUINT EXTENDS ReportableAlarm
  VAR_GLOBAL
    sReportableAlarmMaskReferenceUINT : t_medium_string := 'AlarmMskRefUINT';
  END_VAR
  VAR
    lState : BOOL := FALSE;
    lInputReference : REFERENCE TO UINT;
    lMask : WORD;
  END_VAR

            
          

METHOD describe
  VAR_INPUT
    executeContext : POINTER TO ExecuteContext;
  END_VAR
                  SUPER^.describe(executeContext);

IF (executeContext^.matchOption(cExecuteOptionSyntax)) THEN
	RETURN;
END_IF

IF (executeContext^.matchOption(cExecuteOptionParameter)) THEN	
	RETURN;
END_IF

IF (executeContext^.matchOption(cExecuteOptionVerbose)) THEN	
	executeContext^.appendPair('input',gTypeHandler.getTokenForUINT(lInputReference),FALSE,TRUE);
	executeContext^.appendPair('mask',WORD_TO_STRING(Mask),FALSE,TRUE);
	executeContext^.appendPair('state',gTypeHandler.getTokenForBool(State),FALSE,TRUE);
END_IF



                
END_METHOD

METHOD initialize
                  IF (NOT(__ISVALIDREF(lInputReference))) THEN
	gCodeErrorHandler(pMessage:=CONCAT('null reference in ',lIdentity));
END_IF

SUPER^.initialize();

                
END_METHOD

METHOD initializeStateOp
  VAR_INPUT
    p : POINTER TO t_particle_op;
    name : t_token_string;
    code : t_state_code;
  END_VAR
                  lCode := code;

IF (name='') THEN
	Name := getStringForStateCode(Code);
ELSE
	Name := name;
END_IF

IF (p=0) THEN
	gCodeErrorHandler(pMessage:='initializing reportable with null t_particle_op');
	RETURN;
END_IF

p^.registerOperational(THIS);


                
END_METHOD

METHOD operator
                  lState := WORD_TO_BOOL(lMask AND UINT_TO_WORD(lInputReference));

SUPER^.operator();

IF (lState) THEN
	trigger(FALSE);
END_IF

                
END_METHOD
END_FUNCTION_BLOCK

{attribute 'object_name' := 'ReportableAlarmReferenceUINT'}
FUNCTION_BLOCK ReportableAlarmReferenceUINT EXTENDS ReportableAlarm
  VAR_GLOBAL
    sReportableAlarmReferenceUINT : t_medium_string := 'AlarmMskRefUINT';
  END_VAR
  VAR
    lState : BOOL := FALSE;
    lInputReference : REFERENCE TO UINT;
    lIndex : USINT;
  END_VAR

            
          

METHOD describe
  VAR_INPUT
    executeContext : POINTER TO ExecuteContext;
  END_VAR
                  SUPER^.describe(executeContext);

IF (executeContext^.matchOption(cExecuteOptionSyntax)) THEN
	RETURN;
END_IF

IF (executeContext^.matchOption(cExecuteOptionParameter)) THEN	
	RETURN;
END_IF

executeContext^.appendPair('Severity',gTypeHandler.getTokenForEnum(cEnumTypeSeverity,Severity),TRUE,TRUE);

                
END_METHOD

METHOD initialize
                  IF (NOT(__ISVALIDREF(lInputReference))) THEN
	gCodeErrorHandler(pMessage:=CONCAT('null reference in ',lIdentity));
END_IF

SUPER^.initialize();

                
END_METHOD

METHOD operator
                  lState := fExtractBoolFromWord(UINT_TO_WORD(lInputReference),pStart:=lIndex);

SUPER^.operator();

IF (lState) THEN
	trigger(FALSE);
END_IF

                
END_METHOD
END_FUNCTION_BLOCK

FUNCTION_BLOCK ReportableAlarmSubsystem EXTENDS ReportableAlarm
  VAR
    lSubsystemCode : t_state_code;
  END_VAR

            
          

METHOD describe
  VAR_INPUT
    executeContext : POINTER TO ExecuteContext;
  END_VAR
                  SUPER^.describe(executeContext);

IF (executeContext^.matchOption(cExecuteOptionSyntax)) THEN
	RETURN;
END_IF

IF (executeContext^.matchOption(cExecuteOptionParameter)) THEN	
	RETURN;
END_IF

IF (executeContext^.matchOption(cExecuteOptionVerbose)) THEN	
	executeContext^.appendPair('subsystem_code',getStringForStateCode(SubsystemCode),TRUE,TRUE);
END_IF

                
END_METHOD

PROPERTY SubsystemCode : t_state_code
GET
                    SubsystemCode := lSubsystemCode;

                  
END_GET
SET
                    lSubsystemCode := SubsystemCode;
lContext := INT_TO_LWORD(SubsystemCode);
                  
END_SET
END_PROPERTY

PROPERTY TypeToken : t_medium_string
GET
                    TypeToken := 'AlarmSubsystem';
                  
END_GET
END_PROPERTY
END_FUNCTION_BLOCK

FUNCTION_BLOCK ReportableCausal EXTENDS ReportableState

            
          

PROPERTY TypeToken : t_medium_string
GET
                    TypeToken := 'Causal';
                  
END_GET
END_PROPERTY
END_FUNCTION_BLOCK

FUNCTION_BLOCK ReportableDiagnostic EXTENDS ReportableState

            
          

PROPERTY TypeToken : t_medium_string
GET
                    TypeToken := 'Diagnostic';
                  
END_GET
END_PROPERTY
END_FUNCTION_BLOCK

FUNCTION_BLOCK PersistentStream EXTENDS PersistentValue
  VAR
    lValue : t_stream;
  END_VAR

            
          

METHOD initialize
                  lData := lValue.Buffer;
lCount := lValue.BufferSize;

SUPER^.initialize();

lValue.setLength();


                
END_METHOD

METHOD clear
                  IF (lValue.Length=0) THEN
	RETURN;
END_IF

lValue.clear();
write();
                
END_METHOD

METHOD import
  VAR_INPUT
    stream : REFERENCE TO t_stream;
  END_VAR
                  IF (NOT(__ISVALIDREF(stream))) THEN
	RETURN;	
END_IF

lValue.import(stream);
write();
                
END_METHOD

METHOD export
  VAR_INPUT
    stream : REFERENCE TO t_stream;
  END_VAR
                  IF (NOT(__ISVALIDREF(stream))) THEN
	RETURN;	
END_IF

stream.import(this^);
                
END_METHOD
END_FUNCTION_BLOCK

FUNCTION_BLOCK PersistentStreamStore EXTENDS PersistentValue
  VAR CONSTANT
    cBufferSize : UINT := 24000;
  END_VAR
  VAR
    lValue : ARRAY[0..cBufferSize] OF BYTE;
    lLength : UINT := 0;
  END_VAR

            
          

METHOD initialize
                  lData := ADR(lValue[0]);
lCount := SIZEOF(lValue);

SUPER^.initialize();


                
END_METHOD

METHOD append
                  
                
END_METHOD

METHOD clear
                  lLength := 0;
lValue[0] := 0;
                
END_METHOD
END_FUNCTION_BLOCK

FUNCTION_BLOCK Stream
  VAR CONSTANT
    cBufferSize : UINT := 8187;
    cBufferUseableSize : UINT := 8191;
  END_VAR
  VAR
    lBuffer : ARRAY[0..cBufferSize] OF BYTE;
    lLength : UINT := 0;
    lCharacters : UINT := 0;
    lOverflow : BOOL := FALSE;
    lIndent : t_medium_string;
    lNewline : t_short_string := '$R$N';
    lIndentStr : t_short_string := '    ';
    lRecordInitiator : t_short_string := '{';
    lRecordTerminator : t_short_string := '}$R$N';
    lParsePtr : POINTER TO BYTE := ADR(lBuffer[0]);
    lTerminatorPtr : POINTER TO BYTE := ADR(lBuffer[0]);
    lCurrentToken : t_parse_token_type := cParseTokenNone;
    lParseDebug : BOOL := FALSE;
  END_VAR

            
          

METHOD append
  VAR_INPUT
    str : STRING;
  END_VAR
  VAR
    lng : UINT;
    avail : UINT;
  END_VAR
                  lng := INT_TO_UINT(len(str));
IF (lng=0) THEN
	RETURN;
END_IF

IF (cBufferUseableSize<=lCharacters) THEN
	lOverflow := TRUE;
	RETURN;
END_IF

avail := cBufferUseableSize - lCharacters;

IF (lng>avail) THEN
	lng := avail;
	lOverflow := TRUE;
END_IF

MEMUtils.MemCpy(ADR(lBuffer[lCharacters]),ADR(str[0]),lng+1);

lCharacters := lCharacters + lng;
lLength := lCharacters + 1;
                
END_METHOD

METHOD appendPtr
  VAR_INPUT
    str : POINTER TO t_long_string;
  END_VAR
  VAR
    lng : UINT;
    avail : UINT;
  END_VAR
                  IF (str=0) THEN
	RETURN;
END_IF

lng := INT_TO_UINT(len(str^));
IF (lng=0) THEN
	RETURN;
END_IF

IF (cBufferUseableSize<=lCharacters) THEN
	lOverflow := TRUE;
	RETURN;
END_IF

avail := cBufferUseableSize - lCharacters;

IF (lng>avail) THEN
	lng := avail;
	lOverflow := TRUE;
END_IF

MEMUtils.MemCpy(ADR(lBuffer[lCharacters]),ADR(str^[0]),lng+1);

lCharacters := lCharacters + lng;
lLength := lCharacters + 1;
                
END_METHOD

METHOD checkTermination
                  IF (lLength=0) THEN
	lCharacters := 0;
	lBuffer[0] := 0;
	lTerminatorPtr := ADR(lBuffer[0]);

	RETURN;
END_IF

IF (lBuffer[lLength-1]<>0) THEN
	lBuffer[lLength] := 0;
	lCharacters := lLength;
	lLength := lLength + 1;
ELSE
	lCharacters := lLength - 1;
END_IF

lTerminatorPtr := ADR(lBuffer[lCharacters]);

                
END_METHOD

METHOD clear
                  lLength := 0;
lCharacters := 0;
lBuffer[0] := 0;
lOverflow := FALSE;
lIndent := '';
lParsePtr := ADR(lBuffer[0]);
lTerminatorPtr := ADR(lBuffer[0]);

lCurrentToken := cParseTokenSimple;

                
END_METHOD

METHOD copyToLongString
  VAR_INPUT
    str : POINTER TO t_long_string;
  END_VAR
  VAR
    lng : UINT;
    i : UINT;
  END_VAR
                  IF (str=0) THEN
	RETURN;
END_IF

lng := MIN(lCharacters,63);
lng := lng + 1;

FOR i:=0 TO lng DO
	str^[i] := lBuffer[i];
END_FOR

                
END_METHOD

METHOD decreaseIndent
  VAR
    l : INT;
    i : INT;
  END_VAR
                  l := LEN(lIndent);
i := LEN(lIndentStr);

IF (l<=i) THEN
	lIndent := '';
	RETURN;
END_IF

l := MAX(l-i,i);

lIndent := LEFT(lIndent,l);

                
END_METHOD

METHOD increaseIndent
                  lIndent := CONCAT(lIndent,lIndentStr);
                
END_METHOD

METHOD indent
                  append(lIndent);
                
END_METHOD

METHOD initializeParsing
                  lParsePtr := ADR(lBuffer[0]);
lTerminatorPtr := lParsePtr + lLength;
lCurrentToken := cParseTokenSimple;

                
END_METHOD

METHOD newline
                  append(lNewline);
                
END_METHOD

METHOD getNextToken : t_parse_token_type
  VAR_INPUT
    tokenPtr : POINTER TO t_fqtoken_string;
  END_VAR
  VAR
    c : BYTE;
    length : UINT := 0;
    bytePtr : POINTER TO BYTE;
  END_VAR
                  bytePtr := ADR(tokenPtr^[0]);

IF ((lCurrentToken=cParseTokenError) OR
	(lCurrentToken=cParseTokenOverflow) OR
	(lCurrentToken=cParseTokenFinished)) THEN

	lCurrentToken := cParseTokenFinished;	

	bytePtr^ := 0;
	getNextToken := lCurrentToken;
	parseDebug(getNextToken,tokenPtr);	

	RETURN;	
END_IF

lCurrentToken := cParseTokenSimple;

WHILE (lParsePtr<=lTerminatorPtr) DO
	c := lParsePtr^;

	CASE c OF
		0: // terminator
			IF (length=0) THEN
				lCurrentToken := cParseTokenFinished;
			END_IF
			
			bytePtr^ := 0;
			getNextToken := lCurrentToken;
			parseDebug(getNextToken,tokenPtr);	
			RETURN;
			
		32, // space
		9, // tab
		10, // lf
		11, // vtab
		12, // ff
		13: // cr
			lParsePtr := lParsePtr + 1;
			skipWhiteSpace();

			IF (length>0) THEN
				bytePtr^ := 0;
				getNextToken := lCurrentToken;			
				parseDebug(getNextToken,tokenPtr);		
				RETURN;
			END_IF
			
			CONTINUE;
		
		35: // #
			lParsePtr := lParsePtr + 1;
			skipPastEOL();

			IF (length>0) THEN		
				bytePtr^ := 0;
				getNextToken := lCurrentToken;			
				parseDebug(getNextToken,tokenPtr);		
				RETURN;
			END_IF
			
			CONTINUE;

		44, // ,
		59: // ;

			IF (length>0) THEN				
				bytePtr^ := 0;
				getNextToken := lCurrentToken;			
				parseDebug(getNextToken,tokenPtr);		
				RETURN;
			END_IF
			
			lParsePtr := lParsePtr + 1;
			lCurrentToken := cParseTokenTerminator;

			bytePtr^ := 0;			
			getNextToken := lCurrentToken;			
			parseDebug(getNextToken,tokenPtr);	
			RETURN;			
		
		47: // /
			IF (NOT(lCurrentToken=cParseTokenSimple)) THEN
				lCurrentToken := cParseTokenError;
			ELSIF (length>0) THEN
				lCurrentToken := cParseTokenName;
			ELSE
				lCurrentToken := cParseTokenError;
			END_IF

			lParsePtr := lParsePtr + 1;	

			bytePtr^ := 0;
			getNextToken := lCurrentToken;			
			parseDebug(getNextToken,tokenPtr);		
			RETURN;

		61: // =
			IF (lCurrentToken=cParseTokenOption) THEN
				lCurrentToken := cParseTokenError;
			ELSIF (length>0) THEN
				lCurrentToken := cParseTokenParameter;
			ELSE
				lCurrentToken := cParseTokenError;
			END_IF

			lParsePtr := lParsePtr + 1;	

			bytePtr^ := 0;
			getNextToken := lCurrentToken;			
			parseDebug(getNextToken,tokenPtr);		
			RETURN;
		
		45: // -
			IF (length=0) THEN
				lCurrentToken := cParseTokenOption;
				lParsePtr := lParsePtr + 1;
				CONTINUE;
			END_IF
	END_CASE

	c := lParsePtr^;

	// not alphanumeric	or -_.:
	IF (NOT(((c>=48) AND (c<=57)) OR
		((c>=65) AND (c<=90)) OR
		((c>=97) AND (c<=122)) OR
		(c=45) OR
		(c=46) OR
		(c=58) OR
		(c=95))) THEN
		lParsePtr := lParsePtr + 1;
		CONTINUE;	
	END_IF
				
	IF (length>=INT_TO_UINT(SIZEOF(t_fqtoken_string)-1)) THEN
		lCurrentToken := cParseTokenOverflow;
		
		lParsePtr := lParsePtr + 1;

		bytePtr^ := 0;
		getNextToken := lCurrentToken;			
		parseDebug(getNextToken,tokenPtr);		
		RETURN;
	END_IF
	
	bytePtr^ := lParsePtr^;
	
	bytePtr := bytePtr + 1;
	lParsePtr := lParsePtr + 1;
	length := length + 1;
END_WHILE

IF (length=0) THEN
	lCurrentToken := cParseTokenFinished;
END_IF			

bytePtr^ := 0;
getNextToken := lCurrentToken;			
parseDebug(getNextToken,tokenPtr);		

                
END_METHOD

METHOD parseDebug
  VAR_INPUT
    tokenType : t_parse_token_type;
    tokenPtr : POINTER TO t_token_string;
  END_VAR
                  IF (NOT(lParseDebug)) THEN
	RETURN;
END_IF

append('debug - found token <');
append(tokenPtr^);
append('> of type <');
append(getStringForParseTokenType(tokenType));
append('>');
newline();	

                
END_METHOD

METHOD skipPastEOL
  VAR
    c : BYTE;
  END_VAR
                  WHILE (lParsePtr<lTerminatorPtr) DO
	IF ((lParsePtr^=0) OR
		(lParsePtr^=10) OR
		(lParsePtr^=13)) THEN
		RETURN;
	END_IF
	
	lParsePtr := lParsePtr + 1;
END_WHILE

                
END_METHOD

METHOD skipWhiteSpace
  VAR
    c : BYTE;
  END_VAR
                  WHILE (lParsePtr<lTerminatorPtr) DO
	IF ((lParsePtr^<>32) AND
		(lParsePtr^<9) OR
		(lParsePtr^>13)) THEN
		RETURN;
	END_IF
	
	lParsePtr := lParsePtr + 1;
END_WHILE

                
END_METHOD

METHOD terminateWithNewline
  VAR
    str : t_short_string;
    lng : INT;
  END_VAR
                  str := '$r$n';

MEMUtils.MemCpy(ADR(lBuffer[lCharacters]),ADR(str[0]),3);

lCharacters := lCharacters + 2;
lLength := lCharacters + 1;
                
END_METHOD

METHOD skipOverError
  VAR
    c : BYTE;
  END_VAR
                  WHILE (lParsePtr<lTerminatorPtr) DO
	IF ((lParsePtr^=0) OR
		(lParsePtr^=44) OR
		(lParsePtr^=59) OR
		(lParsePtr^=10) OR
		(lParsePtr^=13)) THEN
		RETURN;
	END_IF
	
	lParsePtr := lParsePtr + 1;
END_WHILE

                
END_METHOD

METHOD recordTerminator
                  append(lRecordTerminator);
                
END_METHOD

METHOD recordInitiator
                  append(lRecordInitiator);
                
END_METHOD

METHOD equals : BOOL
  VAR_INPUT
    stream : REFERENCE TO t_stream;
  END_VAR
                  IF (NOT(__ISVALIDREF(stream))) THEN
	equals := FALSE;
	RETURN;	
END_IF

IF (stream.Length<>Length) THEN
	equals := FALSE;
	RETURN;
END_IF

equals := MEMUtils.MemCmp(stream.Buffer,ADR(lBuffer[0]),UINT_TO_DWORD(lLength));
                
END_METHOD

METHOD import
  VAR_INPUT
    buffer : POINTER TO t_store_buffer;
  END_VAR
                  IF (buffer=0) THEN
	RETURN;	
END_IF

MEMUtils.MemCpy(ADR(lBuffer[0]),buffer,UINT_TO_DWORD(stream.Length));

lLength := stream.Length;
lCharacters := stream.Characters;

                
END_METHOD

